DATA_BLOCK "Error_Safety"	// DB 410
AUTHOR : Koenig
VERSION : 0.1
  STRUCT
   Error_09 : BOOL ;	//Emergency stop door 9
   Error_10 : BOOL ;	//Emergency stop door 10
   Error_11 : BOOL ;	//Emergency stop door 11
   Error_12 : BOOL ;	//Emergency stop door 12
   Error_13 : BOOL ;	//Emergency stop door 13
   Error_14 : BOOL ;	//Emergency stop door 14
   Error_15 : BOOL ;	//Emergency stop door 15
   Error_16 : BOOL ;	//Emergency stop door 16
   Error_01 : BOOL ;	//Emergency stop door 1
   Error_02 : BOOL ;	//Emergency stop door 2
   Error_03 : BOOL ;	//Emergency stop door 3
   Error_04 : BOOL ;	//Emergency stop door 4
   Error_05 : BOOL ;	//Emergency stop door 5
   Error_06 : BOOL ;	//Emergency stop door 6
   Error_07 : BOOL ;	//Emergency stop door 7
   Error_08 : BOOL ;	//Emergency stop door 8
   Error_25 : BOOL ;	//Door 9 is unlocked
   Error_26 : BOOL ;	//Door 10 is unlocked
   Error_27 : BOOL ;	//Door 11 is unlocked
   Error_28 : BOOL ;	//Door 12 is unlocked
   Error_29 : BOOL ;	//Door 13 is unlocked
   Error_30 : BOOL ;	//Door 14 is unlocked
   Error_31 : BOOL ;	//Door 15 is unlocked
   Error_32 : BOOL ;	//Door 16 is unlocked
   Error_17 : BOOL ;	//Door 1 is unlocked
   Error_18 : BOOL ;	//Door 2 is unlocked
   Error_19 : BOOL ;	//Door 3 is unlocked
   Error_20 : BOOL ;	//Door 4 is unlocked
   Error_21 : BOOL ;	//Door 5 is unlocked
   Error_22 : BOOL ;	//Door 6 is unlocked
   Error_23 : BOOL ;	//Door 7 is unlocked
   Error_24 : BOOL ;	//Door 8 is unlocked
   Error_41 : BOOL ;
   Error_42 : BOOL ;
   Error_43 : BOOL ;
   Error_44 : BOOL ;
   Error_45 : BOOL ;
   Error_46 : BOOL ;
   Error_47 : BOOL ;
   Error_48 : BOOL ;
   Error_33 : BOOL ;	//Safety light beam 1 tripped
   Error_34 : BOOL ;	//Safety light beam 2 tripped
   Error_35 : BOOL ;	//Safety light beam 3 tripped
   Error_36 : BOOL ;	//Safety light beam 4 tripped
   Error_37 : BOOL ;	//Safety light beam 5 tripped
   Error_38 : BOOL ;	//Safety light beam 6 tripped
   Error_39 : BOOL ;	//Safety light beam 7 tripped
   Error_40 : BOOL ;	//Safety light beam 8 tripped
   Error_57 : BOOL ;
   Error_58 : BOOL ;
   Error_59 : BOOL ;
   Error_60 : BOOL ;
   Error_61 : BOOL ;
   Error_62 : BOOL ;
   Error_63 : BOOL ;
   Error_64 : BOOL ;
   Error_49 : BOOL ;
   Error_50 : BOOL ;	//Emergency stop master
   Error_51 : BOOL ;	//Emergency stop view station #1
   Error_52 : BOOL ;	//Emergency stop view station #2
   Error_53 : BOOL ;	//Emergency stop view station #3
   Error_54 : BOOL ;	//Emergency stop remote crane 1
   Error_55 : BOOL ;	//Emergency stop remote crane 2
   Error_56 : BOOL ;	//Emergency stop main cabinet
   Error_73 : BOOL ;	//CN2 : Relais error emergency mode
   Error_74 : BOOL ;	//CN2 : Relais error bypass remote
   Error_75 : BOOL ;	//CN2 : Relais error fast stop regulator bridge
   Error_76 : BOOL ;	//CN2 : Relais error fast stop regulator trolley
   Error_77 : BOOL ;	//CN2 : Relais error fast stop regulator lift
   Error_78 : BOOL ;	//CN2 : Relais error fast stop regulator width 1
   Error_79 : BOOL ;	//CN2 : Relais error fast stop regulator width 2
   Error_80 : BOOL ;
   Error_65 : BOOL ;	//CN1 : Relais error emergency mode
   Error_66 : BOOL ;	//CN1 : Relais error bypass remote
   Error_67 : BOOL ;	//CN1 : Relais error fast stop regulator bridge
   Error_68 : BOOL ;	//CN1 : Relais error fast stop regulator trolley
   Error_69 : BOOL ;	//CN1 : Relais error fast stop regulator lift
   Error_70 : BOOL ;	//CN1 : Relais error fast stop regulator width 1
   Error_71 : BOOL ;	//CN1 : Relais error fast stop regulator width 2
   Error_72 : BOOL ;
   Error_89 : BOOL ;	//CN2 : no release fast speed bridge
   Error_90 : BOOL ;	//CN2 : no release bridge
   Error_91 : BOOL ;	//CN2 : no release trolley
   Error_92 : BOOL ;	//CN2 : no release lift
   Error_93 : BOOL ;	//CN2 : no release width 1
   Error_94 : BOOL ;	//CN2 : no release width 2
   Error_95 : BOOL ;	//CN2 : no release safety bar
   Error_96 : BOOL ;
   Error_81 : BOOL ;	//CN1 : no release fast speed bridge
   Error_82 : BOOL ;	//CN1 : no release bridge
   Error_83 : BOOL ;	//CN1 : no release trolley
   Error_84 : BOOL ;	//CN1 : no release lift
   Error_85 : BOOL ;	//CN1 : no release width 1
   Error_86 : BOOL ;	//CN1 : no release width 2
   Error_87 : BOOL ;	//CN1 : no release safety bar
   Error_88 : BOOL ;
   Error_105 : BOOL ;	//CN2 : Invalid safety position
   Error_106 : BOOL ;	//CN2 : Invalid safe speed
   Error_107 : BOOL ;	//CN2 : Invalid max speed
   Error_108 : BOOL ;	//CN2 : Safety position difference
   Error_109 : BOOL ;	//CN2 : Signal fault safety closed
   Error_110 : BOOL ;	//CN2 : Invalid operation mode
   Error_111 : BOOL ;	//CN2 : Emergency mode
   Error_112 : BOOL ;	//CN2 : Brake resistors are not OK
   Error_97 : BOOL ;	//CN1 : Invalid safety position
   Error_98 : BOOL ;	//CN1 : Invalid safe speed
   Error_99 : BOOL ;	//CN1 : Invalid max speed
   Error_100 : BOOL ;	//CN1 : Safety position difference
   Error_101 : BOOL ;	//CN1 : Signal fault safety closed
   Error_102 : BOOL ;	//CN1 : Invalid operation mode
   Error_103 : BOOL ;	//CN1 : Emergency mode
   Error_104 : BOOL ;	//CN1 : Brake resistors are not OK
   Error_121 : BOOL ;	//CN2 : Automatic Mode
   Error_122 : BOOL ;	//CN2 : Bypass active
   Error_123 : BOOL ;	//CN2 : Emergency Mode
   Error_124 : BOOL ;	//CN2 : Maintenance
   Error_125 : BOOL ;	//CN2 : crane not on maintenance position
   Error_126 : BOOL ;
   Error_127 : BOOL ;
   Error_128 : BOOL ;
   Error_113 : BOOL ;	//CN1 : Automatic Mode
   Error_114 : BOOL ;	//CN1 : Bypass active
   Error_115 : BOOL ;	//CN1 : Emergency Mode
   Error_116 : BOOL ;	//CN1 : Maintenance
   Error_117 : BOOL ;	//CN1 : crane not on maintenance position
   Error_118 : BOOL ;
   Error_119 : BOOL ;
   Error_120 : BOOL ;
   Error_137 : BOOL ;	//CN2 : Wago unit #1 disturbed
   Error_138 : BOOL ;	//CN2 : Wago unit #2 disturbed
   Error_139 : BOOL ;	//CN2 : Wago unit #3 disturbed
   Error_140 : BOOL ;	//CN2 : Wago unit #4 disturbed
   Error_141 : BOOL ;	//CN2 : Wago unit #5 disturbed
   Error_142 : BOOL ;
   Error_143 : BOOL ;
   Error_144 : BOOL ;
   Error_129 : BOOL ;	//CN1 : Wago unit #1 disturbed
   Error_130 : BOOL ;	//CN1 : Wago unit #2 disturbed
   Error_131 : BOOL ;	//CN1 : Wago unit #3 disturbed
   Error_132 : BOOL ;	//CN1 : Wago unit #4 disturbed
   Error_133 : BOOL ;	//CN1 : Wago unit #5 disturbed
   Error_134 : BOOL ;
   Error_135 : BOOL ;
   Error_136 : BOOL ;
   Error_153 : BOOL ;	//CB : Wago unit #9 disturbed
   Error_154 : BOOL ;	//CB : Wago unit #10 disturbed
   Error_155 : BOOL ;	//CB : Wago unit #11 disturbed
   Error_156 : BOOL ;	//CB : Wago unit #12 disturbed
   Error_157 : BOOL ;	//CB : Wago unit #13 disturbed
   Error_158 : BOOL ;	//CB : Wago unit #14 disturbed
   Error_159 : BOOL ;	//CB : Wago unit #15 disturbed
   Error_160 : BOOL ;	//CB : Wago unit #16 disturbed
   Error_145 : BOOL ;	//CB : Wago unit #1 disturbed
   Error_146 : BOOL ;	//CB : Wago unit #2 disturbed
   Error_147 : BOOL ;	//CB : Wago unit #3 disturbed
   Error_148 : BOOL ;	//CB : Wago unit #4 disturbed
   Error_149 : BOOL ;	//CB : Wago unit #5 disturbed
   Error_150 : BOOL ;	//CB : Wago unit #6 disturbed
   Error_151 : BOOL ;	//CB : Wago unit #7 disturbed
   Error_152 : BOOL ;	//CB : Wago unit #8 disturbed
   Error_169 : BOOL ;	//CR2 : Wago unit #1 disturbed
   Error_170 : BOOL ;	//CR2 : Wago unit #2 disturbed
   Error_171 : BOOL ;	//CR2 : Wago unit #3 disturbed
   Error_172 : BOOL ;	//CR2 : Wago unit #4 disturbed
   Error_173 : BOOL ;
   Error_174 : BOOL ;
   Error_175 : BOOL ;
   Error_176 : BOOL ;
   Error_161 : BOOL ;	//CR1 : Wago unit #1 disturbed
   Error_162 : BOOL ;	//CR1 : Wago unit #2 disturbed
   Error_163 : BOOL ;	//CR1 : Wago unit #3 disturbed
   Error_164 : BOOL ;	//CR1 : Wago unit #4 disturbed
   Error_165 : BOOL ;
   Error_166 : BOOL ;
   Error_167 : BOOL ;
   Error_168 : BOOL ;
   Error_185 : BOOL ;	//MB1 : Wago unit #1 disturbed
   Error_186 : BOOL ;	//MB1 : Wago unit #2 disturbed
   Error_187 : BOOL ;	//MB1 : Wago unit #3 disturbed
   Error_188 : BOOL ;	//MB1 : Wago unit #4 disturbed
   Error_189 : BOOL ;	//SU1 : Wago unit #1 disturbed
   Error_190 : BOOL ;	//SU1 : Wago unit #2 disturbed
   Error_191 : BOOL ;	//SU2 : Wago unit #1 disturbed
   Error_192 : BOOL ;	//SU2 : Wago unit #2 disturbed
   Error_177 : BOOL ;	//CS1 : Wago unit #1 disturbed
   Error_178 : BOOL ;	//CS1 : Wago unit #2 disturbed
   Error_179 : BOOL ;	//CS1 : Wago unit #3 disturbed
   Error_180 : BOOL ;	//CS1 : Wago unit #4 disturbed
   Error_181 : BOOL ;	//CS1 : Wago unit #5 disturbed
   Error_182 : BOOL ;	//CS1 : Wago unit #6 disturbed
   Error_183 : BOOL ;
   Error_184 : BOOL ;
  END_STRUCT ;	
BEGIN
   Error_07 := TRUE;
   Error_137 := TRUE;
   Error_138 := TRUE;
   Error_139 := TRUE;
   Error_140 := TRUE;
   Error_153 := TRUE;
   Error_161 := TRUE;
   Error_185 := TRUE;
   Error_177 := TRUE;
   Error_178 := TRUE;
   Error_179 := TRUE;
   Error_180 := TRUE;
   Error_181 := TRUE;
END_DATA_BLOCK

// DB 450: know-how protected block, not included

// DB 451: know-how protected block, not included

// DB 545: know-how protected block, not included

// DB 546: know-how protected block, not included

// DB 547: know-how protected block, not included

// DB 548: know-how protected block, not included

// DB 549: know-how protected block, not included

// DB 550: know-how protected block, not included

// DB 551: know-how protected block, not included

// DB 552: know-how protected block, not included

// DB 553: know-how protected block, not included

// DB 554: know-how protected block, not included

// DB 555: know-how protected block, not included

// DB 556: know-how protected block, not included

// DB 557: know-how protected block, not included

// DB 558: know-how protected block, not included

// DB 559: know-how protected block, not included

// DB 560: know-how protected block, not included

// DB 561: know-how protected block, not included

// DB 562: know-how protected block, not included

DATA_BLOCK "F_IO"	// DB 690
AUTHOR : Koenig
VERSION : 0.1
  STRUCT
   BRI_EStop : BOOL ;
   BRI_FB_FastStop : BOOL ;
   BRI_FB_EStop_CH1 : BOOL ;
   BRI_FB_EStop_CH2 : BOOL ;
   BRI_Input_04 : BOOL ;
   BRI_Input_05 : BOOL ;
   BRI_Input_06 : BOOL ;
   BRI_Input_07 : BOOL ;
   BRI_TRO_inParkPos_CH1 : BOOL ;
   BRI_TRO_inParkPos_CH2 : BOOL ;
   BRI_Brake_OK : BOOL ;
   BRI_Input_11 : BOOL ;
   BRI_Input_12 : BOOL ;
   BRI_Input_13 : BOOL ;
   BRI_Input_14 : BOOL ;
   BRI_HardwareOK : BOOL ;
   TRO_Spare_DI_35_0 : BOOL ;
   TRO_Spare_DI_35_1 : BOOL ;
   TRO_FB_FastStop_LIF : BOOL ;
   TRO_FB_FastStop_TRO : BOOL ;
   TRO_FB_TastStop_TEL : BOOL ;
   TRO_Spare_DI_40_1 : BOOL ;
   TRO_FB_Estop_CH1 : BOOL ;
   TRO_FB_Estop_CH2 : BOOL ;
   TRO_EStop : BOOL ;
   TRO_Brakes_OK : BOOL ;
   TRO_Spare_DI_45_2 : BOOL ;
   TRO_Spare_DI_45_3 : BOOL ;
   TRO_Input_12 : BOOL ;
   TRO_Input_13 : BOOL ;
   TRO_Input_14 : BOOL ;
   TRO_HardwareOK : BOOL ;
   LIF_Overl_L_NC : BOOL ;
   LIF_Overl_R_NC : BOOL ;
   LIF_Slap_L_NC : BOOL ;
   LIF_Slap_R_NC : BOOL ;
   LIF_Input_04 : BOOL ;
   LIF_Input_05 : BOOL ;
   LIF_Input_06 : BOOL ;
   LIF_Input_07 : BOOL ;
   LIF_Input_08 : BOOL ;
   LIF_Input_09 : BOOL ;
   LIF_Input_10 : BOOL ;
   LIF_Input_11 : BOOL ;
   LIF_Input_12 : BOOL ;
   LIF_Input_13 : BOOL ;
   LIF_Input_14 : BOOL ;
   LIF_HardwareOK : BOOL ;
   CB1_FastStop_Gate_CH1 : BOOL ;
   CB1_FastStop_Gate_CH2 : BOOL ;
   CB1_SPARE_DI220_2 : BOOL ;
   CB1_SPARE_DI220_3 : BOOL ;
   CB1_SPARE_DI225_0 : BOOL ;
   CB1_FastStop : BOOL ;
   CB1_Mode_Auto : BOOL ;
   CB1_Mode_Service : BOOL ;
   CB1_LS1_Door_CH1 : BOOL ;
   CB1_LS1_Door_CH2 : BOOL ;
   CB1_LS2_Door_CH1 : BOOL ;
   CB1_LS2_Door_CH2 : BOOL ;
   CB1_LS3_Door_CH1 : BOOL ;
   CB1_LS3_Door_CH2 : BOOL ;
   CB1_ServiceDoor1_CH1 : BOOL ;
   CB1_ServiceDoor1_CH2 : BOOL ;
   CB1_ServiceDoor2_CH1 : BOOL ;
   CB1_ServiceDoor2_CH2 : BOOL ;
   CB1_ServiceDoor3_CH1 : BOOL ;
   CB1_ServiceDoor3_CH2 : BOOL ;
   CB1_ServiceDoor4_CH1 : BOOL ;
   CB1_ServiceDoor4_CH2 : BOOL ;
   CB1_EStop_Buttons_CH1 : BOOL ;
   CB1_EStop_Buttons_CH2 : BOOL ;
   CB1_EStop_Doors_CH1 : BOOL ;
   CB1_EStop_Doors_CH2 : BOOL ;
   CB1_Service_CH1 : BOOL ;
   CB1_Service_CH2 : BOOL ;
   CB1_Bypass_CH1 : BOOL ;
   CB1_Bypass_CH2 : BOOL ;
   CB1_Auto_ON : BOOL ;
   CB1_SPARE_DI240_7 : BOOL ;
   CB1_PowerON_1 : BOOL ;
   CB1_PowerON_2 : BOOL ;
   CB1_SPARE_DO220_2 : BOOL ;
   CB1_SPARE_DO220_3 : BOOL ;
   CB1_SPARE_DO225_0 : BOOL ;
   CB1_SPARE_DO225_1 : BOOL ;
   CB1_SPARE_DO225_2 : BOOL ;
   CB1_SPARE_DO225_3 : BOOL ;
   MB1_Power_ON_1 : BOOL ;
   MB1_Power_ON_2 : BOOL ;
   MB1_ESTOP_1 : BOOL ;
   MB1_ESTOP_2 : BOOL ;
   MB1_HardwareOK : BOOL ;
   MB1_FB_Power_ON : BOOL ;
   MB1_INPUT_07 : BOOL ;
   MB1_INPUT_08 : BOOL ;
   SU1_HardwareOK : BOOL ;
   SU1_Scanner_Plus_OK : BOOL ;
   SU1_Scanner_Minus_OK : BOOL ;
   SU1_ReglerPowerON : BOOL ;
   SU1_INPUT_05 : BOOL ;
   SU1_INPUT_06 : BOOL ;
   SU1_INPUT_07 : BOOL ;
   SU1_INPUT_08 : BOOL ;
   SU2_HardwareOK : BOOL ;
   SU2_Scanner_Plus_OK : BOOL ;
   SU2_Scanner_Minus_OK : BOOL ;
   SU2_ReglerPowerON : BOOL ;
   SU2_INPUT_05 : BOOL ;
   SU2_INPUT_06 : BOOL ;
   SU2_INPUT_07 : BOOL ;
   SU2_INPUT_08 : BOOL ;
  END_STRUCT ;	
BEGIN
   BRI_EStop := TRUE;
   BRI_FB_EStop_CH2 := TRUE;
   BRI_Input_04 := TRUE;
   TRO_Brakes_OK := TRUE;
   LIF_Overl_L_NC := TRUE;
   LIF_Overl_R_NC := TRUE;
   LIF_Slap_L_NC := TRUE;
   LIF_Slap_R_NC := TRUE;
   CB1_Mode_Auto := TRUE;
   CB1_EStop_Buttons_CH2 := TRUE;
   CB1_EStop_Doors_CH1 := TRUE;
   CB1_EStop_Doors_CH2 := TRUE;
   CB1_Service_CH1 := TRUE;
   CB1_Service_CH2 := TRUE;
   CB1_Auto_ON := TRUE;
   CB1_SPARE_DI240_7 := TRUE;
   CB1_PowerON_1 := TRUE;
   CB1_PowerON_2 := TRUE;
   CB1_SPARE_DO220_2 := TRUE;
   CB1_SPARE_DO220_3 := TRUE;
   CB1_SPARE_DO225_0 := TRUE;
   CB1_SPARE_DO225_1 := TRUE;
   CB1_SPARE_DO225_2 := TRUE;
   CB1_SPARE_DO225_3 := TRUE;
   MB1_FB_Power_ON := TRUE;
END_DATA_BLOCK

DATA_BLOCK "F_Position"	// DB 695
VERSION : 0.1
  STRUCT
   TR_POS_CM : INT ;
   CAR1_ActualPos : INT ;
   CAR2_ActualPos : INT ;
   TR_POS_CM_REL : INT ;
   Spare02 : INT ;
   BR_Area : INT ;
   TR_Area : INT ;
   Spare03 : INT ;
   Spare04 : INT ;
   Spare05 : INT ;
   BR01_TR0209_Start : INT ;	//2000 - 5000
   BR01_TR0209_Stop : INT ;
   BR02_TR0209_Start : INT ;	//5000 - 8000
   BR02_TR0209_Stop : INT ;
   BR03_TR0209_Start : INT ;	//8000 - 11000
   BR03_TR0209_Stop : INT ;
   BR04_TR0209_Start : INT ;	//11000 - 14000
   BR04_TR0209_Stop : INT ;
   BR05_TR0209_Start : INT ;	//14000 - 17000
   BR05_TR0209_Stop : INT ;
   BR06_TR0209_Start : INT ;	//17000 - 20000
   BR06_TR0209_Stop : INT ;
   BR07_TR0209_Start : INT ;	//20000 - 23000
   BR07_TR0209_Stop : INT ;
   BR08_TR0209_Start : INT ;	//23000 - 26000
   BR08_TR0209_Stop : INT ;
   BR09_TR0209_Start : INT ;	//26000 - 29000
   BR09_TR0209_Stop : INT ;
   BR10_TR0209_Start : INT ;	//29000 - 32000
   BR10_TR0209_Stop : INT ;
   BR11_TR0209_Start : INT ;	//38000 - 39000
   BR11_TR0209_Stop : INT ;
   BR01_TR11_Start : INT ;	//33000 - 34000
   BR01_TR11_Stop : INT ;
   BR02_TR11_Start : INT ;	//34000 - 35000
   BR02_TR11_Stop : INT ;
   BR03_TR11_Start : INT ;	//35000 - 36000
   BR03_TR11_Stop : INT ;
   BR04_TR11_Start : INT ;	//36000 - 37000
   BR04_TR11_Stop : INT ;
   BR05_TR11_Start : INT ;	//37000 - 38000
   BR05_TR11_Stop : INT ;
   BR06_TR11_Start : INT ;	//xxx
   BR06_TR11_Stop : INT ;
   BR07_TR11_Start : INT ;	//xxx
   BR07_TR11_Stop : INT ;
   BR08_TR11_Start : INT ;	//xxx
   BR08_TR11_Stop : INT ;
   BR09_TR11_Start : INT ;	//xxx
   BR09_TR11_Stop : INT ;
   BR10_TR11_Start : INT ;	//xxx
   BR10_TR11_Stop : INT ;
   CAR01_TR01_Start : INT ;	//0 - 1000
   CAR01_TR01_Stop : INT ;
   CAR02_TR10_Start : INT ;	//32000 - 33000
   CAR02_TR10_Stop : INT ;
  END_STRUCT ;	
BEGIN
   TR_POS_CM := 16021;
   TR_POS_CM_REL := 2401;
   BR_Area := 5;
   TR_Area := 8;
   BR01_TR0209_Start := 1800;
   BR01_TR0209_Stop := 4500;
   BR02_TR0209_Start := 4800;
   BR02_TR0209_Stop := 7500;
   BR03_TR0209_Start := 7800;
   BR03_TR0209_Stop := 10500;
   BR04_TR0209_Start := 10800;
   BR04_TR0209_Stop := 13500;
   BR05_TR0209_Start := 13800;
   BR05_TR0209_Stop := 16500;
   BR06_TR0209_Start := 16800;
   BR06_TR0209_Stop := 19500;
   BR07_TR0209_Start := 19800;
   BR07_TR0209_Stop := 22500;
   BR08_TR0209_Start := 22800;
   BR08_TR0209_Stop := 25500;
   BR09_TR0209_Start := 25800;
   BR09_TR0209_Stop := 28500;
   BR10_TR0209_Start := 28800;
   BR10_TR0209_Stop := 31500;
   CAR01_TR01_Stop := 1000;
   CAR02_TR10_Start := 31900;
   CAR02_TR10_Stop := 32380;
END_DATA_BLOCK

DATA_BLOCK "F_GBL_RECV"	// DB 750
AUTHOR : Koenig
FAMILY : COM_DBS7
VERSION : 0.1
  STRUCT
   Signal01 : BOOL ;	//Automatic mode
   Signal02 : BOOL ;	//Bypass
   Signal03 : BOOL ;	//Reset
   Signal04 : BOOL ;	//NO E-Stop
   Signal05 : BOOL ;	//Start Automatic
   Signal06 : BOOL ;	//Release drive
   Signal07 : BOOL ;	//Release drive fast
   Signal08 : BOOL ;	//Service mode
   Signal09 : BOOL ;
   Signal10 : BOOL ;	//Safety area rack OK
   Signal11 : BOOL ;
   Signal12 : BOOL ;
   Signal13 : BOOL ;
   Signal14 : BOOL ;
   Signal15 : BOOL ;
   Signal16 : BOOL ;
   Signal17 : BOOL ;
   Signal18 : BOOL ;
   Signal19 : BOOL ;
   Signal20 : BOOL ;
   Signal21 : BOOL ;
   Signal22 : BOOL ;
   Signal23 : BOOL ;
   Signal24 : BOOL ;
   Signal25 : BOOL ;
   Signal26 : BOOL ;
   Signal27 : BOOL ;
   Signal28 : BOOL ;
   Signal29 : BOOL ;
   Signal30 : BOOL ;
   Signal31 : BOOL ;
   Signal32 : BOOL ;
   Value01 : INT ;	//Position carrier 1
   Value02 : INT ;	//Position carrier 2
   Value03 : INT ;
   Value04 : INT ;
  END_STRUCT ;	
BEGIN
   Signal01 := TRUE;
   Signal04 := TRUE;
   Signal06 := TRUE;
   Signal07 := TRUE;
   Signal10 := TRUE;
   Value01 := 5;
   Value02 := 3;
END_DATA_BLOCK

// DB 751: know-how protected block, not included

DATA_BLOCK "F_GBL_SEND"	// DB 752
AUTHOR : Koenig
FAMILY : COM_DBS7
VERSION : 0.1
  STRUCT
   Signal01 : BOOL ;	//Trolley is in position (unsafe)
   Signal02 : BOOL ;	//Teleskope is in center (unsafe)
   Signal03 : BOOL ;	//Teleskope is in rear (unsafe)
   Signal04 : BOOL ;	//Teleskope is in front (unsafe)
   Signal05 : BOOL ;	//Lift in top position (unsafe)
   Signal06 : BOOL ;	//Lift in over position (unsafe)
   Signal07 : BOOL ;	//Lift in under position (unsafe)
   Signal08 : BOOL ;	//Lift in top position (unsafe, sensor)
   Signal09 : BOOL ;
   Signal10 : BOOL ;
   Signal11 : BOOL ;
   Signal12 : BOOL ;
   Signal13 : BOOL ;
   Signal14 : BOOL ;
   Signal15 : BOOL ;
   Signal16 : BOOL ;
   Value01 : INT ;	//Area Trolley (no.)
   Value02 : INT ;	//Area Lift (no.)
   Value03 : INT ;	//Area Bridge (no.)
   Value04 : INT ;	//Trolley Axis value
   Value05 : INT ;	//Trolley Axis releative 2-9 / 11
  END_STRUCT ;	
BEGIN
   Signal01 := TRUE;
   Signal02 := TRUE;
   Value01 := 8;
   Value02 := 6;
   Value03 := 5;
   Value04 := 16021;
   Value05 := 2401;
END_DATA_BLOCK

// DB 753: know-how protected block, not included

DATA_BLOCK "IDB_Axis_Position"	// DB 800
AUTHOR : BRO
VERSION : 0.1
"Axis_Position"
BEGIN
END_DATA_BLOCK

DATA_BLOCK "IDB_WagoiPar_Rack"	// DB 901
AUTHOR : JPR
FAMILY : WAGOiPar
VERSION : 0.0
"WAGO_iPar_UDL_4_Mod"
BEGIN
END_DATA_BLOCK

DATA_BLOCK "IDB_WagoiPar_BRI"	// DB 920
AUTHOR : JPR
FAMILY : WAGOiPar
VERSION : 0.0
"WAGO_iPar_UDL_4_Mod"
BEGIN
END_DATA_BLOCK

DATA_BLOCK "IDB_WagoiPar_TRO"	// DB 921
AUTHOR : JPR
FAMILY : WAGOiPar
VERSION : 0.0
"WAGO_iPar_UDL_4_Mod"
BEGIN
END_DATA_BLOCK

DATA_BLOCK "IDB_WagoiPar_LIF"	// DB 922
AUTHOR : JPR
FAMILY : WAGOiPar
VERSION : 0.0
"WAGO_iPar_UDL_4_Mod"
BEGIN
END_DATA_BLOCK

DATA_BLOCK "DB_iPar_Diag"	// DB 930
AUTHOR : JPR
FAMILY : WAGOiPar
VERSION : 0.0
"DiagPROFIsafe_V2_iPar"
BEGIN
END_DATA_BLOCK

DATA_BLOCK "DIAG_PROFI_V2_iPar"	// DB 931
TITLE = Vorlage Datenbaustein zur Ablage der Diagnosedaten FB101
//Template data block used in combination with FB101
//
AUTHOR : JPR
FAMILY : WAGOiPar
NAME : iParInfD
VERSION : 1.0
  STRUCT
   versionInfo_1 : INT  := 101;	//version info main
   versionInfo_2 : WORD  := W#16#100;	//version info release
   spare_4 : WORD ;
   fctReqTimeout : INT  := 6000;	//function request timeout (default 6000; av.cycle plc 5 ms - timeout 30 s)
   dsvLength : INT  := 20;	//lenght of storage data
   maxModules : INT  := 1;	//amount PROFIsafe modules FB101
   adr_module_1 : INT ;	//I/O address module 1
   adr_module_2 : INT ;	//I/O address module 2
   adr_module_3 : INT ;	//I/O address module 3
   adr_module_4 : INT ;	//I/O address module 4
   adr_module_5 : INT ;	//I/O address module 5
   adr_module_6 : INT ;	//I/O address module 6
   adr_module_7 : INT ;	//I/O address module 7
   adr_module_8 : INT ;	//I/O address module 8
   adr_module_9 : INT ;	//I/O address module 9
   adr_module_10 : INT ;	//I/O address module 10
   adr_module_11 : INT ;	//I/O address module 11
   adr_module_12 : INT ;	//I/O address module 12
   spare_34 : WORD ;
   spare_36 : WORD ;
   Init_Date : DATE ;	//startup date application slave
   InitTime : TIME_OF_DAY ;	//startup time application slave
   spare_46 : WORD ;
   spare_48 : WORD ;
   actDateCyle1 : DATE ;	//actual system date of cycle
   actTimeCyle1 : TIME_OF_DAY ;	//actual system time of cycle
   spare_56 : WORD ;
   spare_58 : WORD ;
   QBAD_moduleActive : DWORD ;	//info QBAD at PROFIsafe module active
   ACK_REQ_moduleActive : DWORD ;	//info ACK_REQ at PROFIsafe module active
   READ_DIAG_REQ_module : DWORD ;	//info READ_DIAG_REQ at PROFIsafe module active
   spare_72 : WORD ;
   spare_74 : WORD ;
   check_cfg_done : DWORD ;	//info check cfg done
   read_diag_done : DWORD ;	//info read diag done
   spare_84 : WORD ;
   spare_86 : WORD ;
   resFctReq_ok : DWORD ;	//response function request ok - "bit per module"
   resFctReq_error : DWORD ;	//response function request error - "bit per module"
   spare_96 : WORD ;
   spare_98 : WORD ;
   cmdCtrl_FB101_1 : WORD ;	//cmd / ctrl information FB101
   comCountStart_1 : WORD ;	//comCountStart indication 1
   mod_type_1 : WORD ;	//module type 1
   mod_version_1 : WORD ;	//module version 1
   spare_108 : WORD ;
   state_SFB52_1 : DWORD ;	//state SFB52 module 1
   spare_114 : WORD ;
   spare_116 : WORD ;
   error_date_mod_1 : DATE ;	//error date module 1
   error_time_mod_1 : TIME_OF_DAY ;	//error time module 1
   error_info_mod_1 : WORD ;	//error info read values module 1
   error_F_Module_mod_1 : WORD ;	//error safety module module 1
   error_F_DI_1_mod_1 : WORD ;	//error safety input 1 module 1
   error_F_DI_2_mod_1 : WORD ;	//error safety input 2 module 1
   error_F_DI_3_mod_1 : WORD ;	//error safety input 3 module 1
   error_F_DI_4_mod_1 : WORD ;	//error safety input 4 module 1
   error_F_DI_5_mod_1 : WORD ;	//error safety input 5 module 1
   error_F_DI_6_mod_1 : WORD ;	//error safety input 6 module 1
   error_F_DI_7_mod_1 : WORD ;	//error safety input 7 module 1
   error_F_DI_8_mod_1 : WORD ;	//error safety input 8 module 1
   error_F_DO_1_mod_1 : WORD ;	//error safety output 1 module 1
   error_F_DO_2_mod_1 : WORD ;	//error safety output 2 module 1
   error_F_DO_3_mod_1 : WORD ;	//error safety output 3 module 1
   error_F_DO_4_mod_1 : WORD ;	//error safety output 4 module 1
   error_F_Mod_R48_mod_1 : WORD ;	//error safety R48 module 1
   error_F_Mod_R49_mod_1 : WORD ;	//error safety R49 module 1
   error_F_Mod_R50_mod_1 : WORD ;	//error safety R50 module 1
   error_F_Mod_R51_mod_1 : WORD ;	//error safety R51 module 1
   error_F_Mod_R52_mod_1 : WORD ;	//error safety R52 module 1
   error_F_Mod_R53_mod_1 : WORD ;	//error safety R53 module 1
   error_F_Mod_R54_mod_1 : WORD ;	//error safety R54 module 1
   error_F_Mod_R55_mod_1 : WORD ;	//error safety R55 module 1
   F_Per_DB_B3_mod_1 : WORD ;	//state F-Periphery DB module 1
   spare_170 : WORD ;
   spare_172 : WORD ;
   spare_174 : WORD ;
   spare_176 : WORD ;
   spare_178 : WORD ;
   cmdCtrl_FB101_2 : WORD ;	//cmd / ctrl information FB101
   comCountStart_2 : WORD ;	//comCountStart indication
   mod_type_2 : WORD ;	//module type
   mod_version_2 : WORD ;	//module version
   spare_188 : WORD ;
   state_SFB52_2 : DWORD ;	//state SFB52 module
   spare_194 : WORD ;
   spare_196 : WORD ;
   error_date_mod_2 : DATE ;	//error date module 2
   error_time_mod_2 : TIME_OF_DAY ;	//error time module 2
   error_info_mod_2 : WORD ;	//error info read values module 2
   error_F_Module_mod_2 : WORD ;	//error safety module module 2
   error_F_DI_1_mod_2 : WORD ;	//error safety input 1 module 2
   error_F_DI_2_mod_2 : WORD ;	//error safety input 2 module 2
   error_F_DI_3_mod_2 : WORD ;	//error safety input 3 module 2
   error_F_DI_4_mod_2 : WORD ;	//error safety input 4 module 2
   error_F_DI_5_mod_2 : WORD ;	//error safety input 5 module 2
   error_F_DI_6_mod_2 : WORD ;	//error safety input 6 module 2
   error_F_DI_7_mod_2 : WORD ;	//error safety input 7 module 2
   error_F_DI_8_mod_2 : WORD ;	//error safety input 8 module 2
   error_F_DO_1_mod_2 : WORD ;	//error safety output 1 module 2
   error_F_DO_2_mod_2 : WORD ;	//error safety output 2 module 2
   error_F_DO_3_mod_2 : WORD ;	//error safety output 3 module 2
   error_F_DO_4_mod_2 : WORD ;	//error safety output 4 module 2
   error_F_Mod_R48_mod_2 : WORD ;	//error safety R48 module 2
   error_F_Mod_R49_mod_2 : WORD ;	//error safety R49 module 2
   error_F_Mod_R50_mod_2 : WORD ;	//error safety R50 module 2
   error_F_Mod_R51_mod_2 : WORD ;	//error safety R51 module 2
   error_F_Mod_R52_mod_2 : WORD ;	//error safety R52 module 2
   error_F_Mod_R53_mod_2 : WORD ;	//error safety R53 module 2
   error_F_Mod_R54_mod_2 : WORD ;	//error safety R54 module 2
   error_F_Mod_R55_mod_2 : WORD ;	//error safety R55 module 2
   F_Per_DB_B3_mod_2 : WORD ;	//state F-Periphery DB module 2
   spare_250 : WORD ;
   spare_252 : WORD ;
   spare_254 : WORD ;
   spare_256 : WORD ;
   spare_258 : WORD ;
   cmdCtrl_FB101_3 : WORD ;	//cmd / ctrl information FB101
   comCountStart_3 : WORD ;	//comCountStart indication
   mod_type_3 : WORD ;	//module type
   mod_version_3 : WORD ;	//module version
   spare_268 : WORD ;
   state_SFB52_3 : DWORD ;	//state SFB52 module
   spare_274 : WORD ;
   spare_276 : WORD ;
   error_date_mod_3 : DATE ;	//error date module 3
   error_time_mod_3 : TIME_OF_DAY ;	//error time module 3
   error_info_mod_3 : WORD ;	//error info read values module 3
   error_F_Module_mod_3 : WORD ;	//error safety module module 3
   error_F_DI_1_mod_3 : WORD ;	//error safety input 1 module 3
   error_F_DI_2_mod_3 : WORD ;	//error safety input 2 module 3
   error_F_DI_3_mod_3 : WORD ;	//error safety input 3 module 3
   error_F_DI_4_mod_3 : WORD ;	//error safety input 4 module 3
   error_F_DI_5_mod_3 : WORD ;	//error safety input 5 module 3
   error_F_DI_6_mod_3 : WORD ;	//error safety input 6 module 3
   error_F_DI_7_mod_3 : WORD ;	//error safety input 7 module 3
   error_F_DI_8_mod_3 : WORD ;	//error safety input 8 module 3
   error_F_DO_1_mod_3 : WORD ;	//error safety output 1 module 3
   error_F_DO_2_mod_3 : WORD ;	//error safety output 2 module 3
   error_F_DO_3_mod_3 : WORD ;	//error safety output 3 module 3
   error_F_DO_4_mod_3 : WORD ;	//error safety output 4 module 3
   error_F_Mod_R48_mod_3 : WORD ;	//error safety R48 module 3
   error_F_Mod_R49_mod_3 : WORD ;	//error safety R49 module 3
   error_F_Mod_R50_mod_3 : WORD ;	//error safety R50 module 3
   error_F_Mod_R51_mod_3 : WORD ;	//error safety R51 module 3
   error_F_Mod_R52_mod_3 : WORD ;	//error safety R52 module 3
   error_F_Mod_R53_mod_3 : WORD ;	//error safety R53 module 3
   error_F_Mod_R54_mod_3 : WORD ;	//error safety R54 module 3
   error_F_Mod_R55_mod_3 : WORD ;	//error safety R55 module 3
   F_Per_DB_B3_mod_3 : WORD ;	//state F-Periphery DB module 3
   spare_330 : WORD ;
   spare_332 : WORD ;
   spare_334 : WORD ;
   spare_336 : WORD ;
   spare_338 : WORD ;
   cmdCtrl_FB101_4 : WORD ;	//cmd / ctrl information FB101
   comCountStart_4 : WORD ;	//comCountStart indication
   mod_type4 : WORD ;	//module type
   mod_version_4 : WORD ;	//module version
   spare_348 : WORD ;
   state_SFB52_4 : DWORD ;	//state SFB52 module
   spare_354 : WORD ;
   spare_356 : WORD ;
   error_date_mod_4 : DATE ;	//error date module 4
   error_time_mod_4 : TIME_OF_DAY ;	//error time module 4
   error_info_mod_4 : WORD ;	//error info read values module 4
   error_F_Module_mod_4 : WORD ;	//error safety module module 4
   error_F_DI_1_mod_4 : WORD ;	//error safety input 1 module 4
   error_F_DI_2_mod_4 : WORD ;	//error safety input 2 module 4
   error_F_DI_3_mod_4 : WORD ;	//error safety input 3 module 4
   error_F_DI_4_mod_4 : WORD ;	//error safety input 4 module 4
   error_F_DI_5_mod_4 : WORD ;	//error safety input 5 module 4
   error_F_DI_6_mod_4 : WORD ;	//error safety input 6 module 4
   error_F_DI_7_mod_4 : WORD ;	//error safety input 7 module 4
   error_F_DI_8_mod_4 : WORD ;	//error safety input 8 module 4
   error_F_DO_1_mod_4 : WORD ;	//error safety output 1 module 4
   error_F_DO_2_mod_4 : WORD ;	//error safety output 2 module 4
   error_F_DO_3_mod_4 : WORD ;	//error safety output 3 module 4
   error_F_DO_4_mod_4 : WORD ;	//error safety output 4 module 4
   error_F_Mod_R48_mod_4 : WORD ;	//error safety R48 module 4
   error_F_Mod_R49_mod_4 : WORD ;	//error safety R49 module 4
   error_F_Mod_R50_mod_4 : WORD ;	//error safety R50 module 4
   error_F_Mod_R51_mod_4 : WORD ;	//error safety R51 module 4
   error_F_Mod_R52_mod_4 : WORD ;	//error safety R52 module 4
   error_F_Mod_R53_mod_4 : WORD ;	//error safety R53 module 4
   error_F_Mod_R54_mod_4 : WORD ;	//error safety R54 module 4
   error_F_Mod_R55_mod_4 : WORD ;	//error safety R55 module 4
   F_Per_DB_B3_mod_4 : WORD ;	//state F-Periphery DB module 4
   spare_410 : WORD ;
   spare_412 : WORD ;
   spare_414 : WORD ;
   spare_416 : WORD ;
   spare_418 : WORD ;
   cmdCtrl_FB101_5 : WORD ;	//cmd / ctrl information FB101
   comCountStart_5 : WORD ;	//comCountStart indication
   mod_type_5 : WORD ;	//module type
   mod_version_5 : WORD ;	//module version
   spare_428 : WORD ;
   state_SFB52_5 : DWORD ;	//state SFB52 module
   spare_434 : WORD ;
   spare_436 : WORD ;
   error_date_mod_5 : DATE ;	//error date module 5
   error_time_mod_5 : TIME_OF_DAY ;	//error time module 5
   error_info_mod_5 : WORD ;	//error info read values module 5
   error_F_Module_mod_5 : WORD ;	//error safety module module 5
   error_F_DI_1_mod_5 : WORD ;	//error safety input 1 module 5
   error_F_DI_2_mod_5 : WORD ;	//error safety input 2 module 5
   error_F_DI_3_mod_5 : WORD ;	//error safety input 3 module 5
   error_F_DI_4_mod_5 : WORD ;	//error safety input 4 module 5
   error_F_DI_5_mod_5 : WORD ;	//error safety input 5 module 5
   error_F_DI_6_mod_5 : WORD ;	//error safety input 6 module 5
   error_F_DI_7_mod_5 : WORD ;	//error safety input 7 module 5
   error_F_DI_8_mod_5 : WORD ;	//error safety input 8 module 5
   error_F_DO_1_mod_5 : WORD ;	//error safety output 1 module 5
   error_F_DO_2_mod_5 : WORD ;	//error safety output 2 module 5
   error_F_DO_3_mod_5 : WORD ;	//error safety output 3 module 5
   error_F_DO_4_mod_5 : WORD ;	//error safety output 4 module 5
   error_F_Mod_R48_mod_5 : WORD ;	//error safety R48 module 5
   error_F_Mod_R49_mod_5 : WORD ;	//error safety R49 module 5
   error_F_Mod_R50_mod_5 : WORD ;	//error safety R50 module 5
   error_F_Mod_R51_mod_5 : WORD ;	//error safety R51 module 5
   error_F_Mod_R52_mod_5 : WORD ;	//error safety R52 module 5
   error_F_Mod_R53_mod_5 : WORD ;	//error safety R53 module 5
   error_F_Mod_R54_mod_5 : WORD ;	//error safety R54 module 5
   error_F_Mod_R55_mod_5 : WORD ;	//error safety R55 module 5
   F_Per_DB_B3_mod_5 : WORD ;	//state F-Periphery DB module 5
   spare_490 : WORD ;
   spare_492 : WORD ;
   spare_494 : WORD ;
   spare_496 : WORD ;
   spare_498 : WORD ;
   cmdCtrl_FB101_6 : WORD ;	//cmd / ctrl information FB101
   comCountStart_6 : WORD ;	//comCountStart indication
   mod_type_6 : WORD ;	//module type
   mod_version_6 : WORD ;	//module version
   spare_508 : WORD ;
   state_SFB52_6 : DWORD ;	//state SFB52 module
   spare_514 : WORD ;
   spare_516 : WORD ;
   error_date_mod_6 : DATE ;	//error date module 6
   error_time_mod_6 : TIME_OF_DAY ;	//error time module 6
   error_info_mod_6 : WORD ;	//error info read values module 6
   error_F_Module_mod_6 : WORD ;	//error safety module module 6
   error_F_DI_1_mod_6 : WORD ;	//error safety input 1 module 6
   error_F_DI_2_mod_6 : WORD ;	//error safety input 2 module 6
   error_F_DI_3_mod_6 : WORD ;	//error safety input 3 module 6
   error_F_DI_4_mod_6 : WORD ;	//error safety input 4 module 6
   error_F_DI_5_mod_6 : WORD ;	//error safety input 5 module 6
   error_F_DI_6_mod_6 : WORD ;	//error safety input 6 module 6
   error_F_DI_7_mod_6 : WORD ;	//error safety input 7 module 6
   error_F_DI_8_mod_6 : WORD ;	//error safety input 8 module 6
   error_F_DO_1_mod_6 : WORD ;	//error safety output 1 module 6
   error_F_DO_2_mod_6 : WORD ;	//error safety output 2 module 6
   error_F_DO_3_mod_6 : WORD ;	//error safety output 3 module 6
   error_F_DO_4_mod_6 : WORD ;	//error safety output 4 module 6
   error_F_Mod_R48_mod_6 : WORD ;	//error safety R48 module 6
   error_F_Mod_R49_mod_6 : WORD ;	//error safety R49 module 6
   error_F_Mod_R50_mod_6 : WORD ;	//error safety R50 module 6
   error_F_Mod_R51_mod_6 : WORD ;	//error safety R51 module 6
   error_F_Mod_R52_mod_6 : WORD ;	//error safety R52 module 6
   error_F_Mod_R53_mod_6 : WORD ;	//error safety R53 module 6
   error_F_Mod_R54_mod_6 : WORD ;	//error safety R54 module 6
   error_F_Mod_R55_mod_6 : WORD ;	//error safety R55 module 6
   F_Per_DB_B3_mod_6 : WORD ;	//state F-Periphery DB module 6
   spare_570 : WORD ;
   spare_572 : WORD ;
   spare_574 : WORD ;
   spare_576 : WORD ;
   spare_578 : WORD ;
   cmdCtrl_FB101_7 : WORD ;	//cmd / ctrl information FB101
   comCountStart_7 : WORD ;	//comCountStart indication
   mod_type_7 : WORD ;	//module type
   mod_version_7 : WORD ;	//module version
   spare_588 : WORD ;
   state_SFB52_7 : DWORD ;	//state SFB52 module
   spare_594 : WORD ;
   spare_596 : WORD ;
   error_date_mod_7 : DATE ;	//error date module 7
   error_time_mod_7 : TIME_OF_DAY ;	//error time module 7
   error_info_mod_7 : WORD ;	//error info read values module 7
   error_F_Module_mod_7 : WORD ;	//error safety module module 7
   error_F_DI_1_mod_7 : WORD ;	//error safety input 1 module 7
   error_F_DI_2_mod_7 : WORD ;	//error safety input 2 module 7
   error_F_DI_3_mod_7 : WORD ;	//error safety input 3 module 7
   error_F_DI_4_mod_7 : WORD ;	//error safety input 4 module 7
   error_F_DI_5_mod_7 : WORD ;	//error safety input 5 module 7
   error_F_DI_6_mod_7 : WORD ;	//error safety input 6 module 7
   error_F_DI_7_mod_7 : WORD ;	//error safety input 7 module 7
   error_F_DI_8_mod_7 : WORD ;	//error safety input 8 module 7
   error_F_DO_1_mod_7 : WORD ;	//error safety output 1 module 7
   error_F_DO_2_mod_7 : WORD ;	//error safety output 2 module 7
   error_F_DO_3_mod_7 : WORD ;	//error safety output 3 module 7
   error_F_DO_4_mod_7 : WORD ;	//error safety output 4 module 7
   error_F_Mod_R48_mod_7 : WORD ;	//error safety R48 module 7
   error_F_Mod_R49_mod_7 : WORD ;	//error safety R49 module 7
   error_F_Mod_R50_mod_7 : WORD ;	//error safety R50 module 7
   error_F_Mod_R51_mod_7 : WORD ;	//error safety R51 module 7
   error_F_Mod_R52_mod_7 : WORD ;	//error safety R52 module 7
   error_F_Mod_R53_mod_7 : WORD ;	//error safety R53 module 7
   error_F_Mod_R54_mod_7 : WORD ;	//error safety R54 module 7
   error_F_Mod_R55_mod_7 : WORD ;	//error safety R55 module 7
   F_Per_DB_B3_mod_7 : WORD ;	//state F-Periphery DB module 7
   spare_650 : WORD ;
   spare_652 : WORD ;
   spare_654 : WORD ;
   spare_656 : WORD ;
   spare_658 : WORD ;
   cmdCtrl_FB101_8 : WORD ;	//cmd / ctrl information FB101
   comCountStart_8 : WORD ;	//comCountStart indication
   mod_type_8 : WORD ;	//module type
   mod_version_8 : WORD ;	//module version
   spare_668 : WORD ;
   state_SFB52_8 : DWORD ;	//state SFB52 module
   spare_674 : WORD ;
   spare_676 : WORD ;
   error_date_mod_8 : DATE ;	//error date module 8
   error_time_mod_8 : TIME_OF_DAY ;	//error time module 8
   error_info_mod_8 : WORD ;	//error info read values module 8
   error_F_Module_mod_8 : WORD ;	//error safety module module 8
   error_F_DI_1_mod_8 : WORD ;	//error safety input 1 module 8
   error_F_DI_2_mod_8 : WORD ;	//error safety input 2 module 8
   error_F_DI_3_mod_8 : WORD ;	//error safety input 3 module 8
   error_F_DI_4_mod_8 : WORD ;	//error safety input 4 module 8
   error_F_DI_5_mod_8 : WORD ;	//error safety input 5 module 8
   error_F_DI_6_mod_8 : WORD ;	//error safety input 6 module 8
   error_F_DI_7_mod_8 : WORD ;	//error safety input 7 module 8
   error_F_DI_8_mod_8 : WORD ;	//error safety input 8 module 8
   error_F_DO_1_mod_8 : WORD ;	//error safety output 1 module 8
   error_F_DO_2_mod_8 : WORD ;	//error safety output 2 module 8
   error_F_DO_3_mod_8 : WORD ;	//error safety output 3 module 8
   error_F_DO_4_mod_8 : WORD ;	//error safety output 4 module 8
   error_F_Mod_R48_mod_8 : WORD ;	//error safety R48 module 8
   error_F_Mod_R49_mod_8 : WORD ;	//error safety R49 module 8
   error_F_Mod_R50_mod_8 : WORD ;	//error safety R50 module 8
   error_F_Mod_R51_mod_8 : WORD ;	//error safety R51 module 8
   error_F_Mod_R52_mod_8 : WORD ;	//error safety R52 module 8
   error_F_Mod_R53_mod_8 : WORD ;	//error safety R53 module 8
   error_F_Mod_R54_mod_8 : WORD ;	//error safety R54 module 8
   error_F_Mod_R55_mod_8 : WORD ;	//error safety R55 module 8
   F_Per_DB_B3_mod_8 : WORD ;	//state F-Periphery DB module 8
   spare_730 : WORD ;
   spare_732 : WORD ;
   spare_734 : WORD ;
   spare_736 : WORD ;
   spare_738 : WORD ;
   cmdCtrl_FB101_9 : WORD ;	//cmd / ctrl information FB101
   comCountStart_9 : WORD ;	//comCountStart indication
   mod_type_9 : WORD ;	//module type
   mod_version_9 : WORD ;	//module version
   spare_748 : WORD ;
   state_SFB52_9 : DWORD ;	//state SFB52 module
   spare_754 : WORD ;
   spare_756 : WORD ;
   error_date_mod_9 : DATE ;	//error date module 9
   error_time_mod_9 : TIME_OF_DAY ;	//error time module 9
   error_info_mod_9 : WORD ;	//error info read values module 9
   error_F_Module_mod_9 : WORD ;	//error safety module module 9
   error_F_DI_1_mod_9 : WORD ;	//error safety input 1 module 9
   error_F_DI_2_mod_9 : WORD ;	//error safety input 2 module 9
   error_F_DI_3_mod_9 : WORD ;	//error safety input 3 module 9
   error_F_DI_4_mod_9 : WORD ;	//error safety input 4 module 9
   error_F_DI_5_mod_9 : WORD ;	//error safety input 5 module 9
   error_F_DI_6_mod_9 : WORD ;	//error safety input 6 module 9
   error_F_DI_7_mod_9 : WORD ;	//error safety input 7 module 9
   error_F_DI_8_mod_9 : WORD ;	//error safety input 8 module 9
   error_F_DO_1_mod_9 : WORD ;	//error safety output 1 module 9
   error_F_DO_2_mod_9 : WORD ;	//error safety output 2 module 9
   error_F_DO_3_mod_9 : WORD ;	//error safety output 3 module 9
   error_F_DO_4_mod_9 : WORD ;	//error safety output 4 module 9
   error_F_Mod_R48_mod_9 : WORD ;	//error safety R48 module 9
   error_F_Mod_R49_mod_9 : WORD ;	//error safety R49 module 9
   error_F_Mod_R50_mod_9 : WORD ;	//error safety R50 module 9
   error_F_Mod_R51_mod_9 : WORD ;	//error safety R51 module 9
   error_F_Mod_R52_mod_9 : WORD ;	//error safety R52 module 9
   error_F_Mod_R53_mod_9 : WORD ;	//error safety R53 module 9
   error_F_Mod_R54_mod_9 : WORD ;	//error safety R54 module 9
   error_F_Mod_R55_mod_9 : WORD ;	//error safety R55 module 9
   F_Per_DB_B3_mod_9 : WORD ;	//state F-Periphery DB module 9
   spare_810 : WORD ;
   spare_812 : WORD ;
   spare_814 : WORD ;
   spare_816 : WORD ;
   spare_818 : WORD ;
   cmdCtrl_FB101_10 : WORD ;	//cmd / ctrl information FB101
   comCountStart_10 : WORD ;	//comCountStart indication
   mod_type_10 : WORD ;	//module type
   mod_version_10 : WORD ;	//module version
   spare_828 : WORD ;
   state_SFB52_10 : DWORD ;	//state SFB52 module
   spare_834 : WORD ;
   spare_836 : WORD ;
   error_date_mod_10 : DATE ;	//error date module 10
   error_time_mod_10 : TIME_OF_DAY ;	//error time module 10
   error_info_mod_10 : WORD ;	//error info read values module 10
   error_F_Module_mod_10 : WORD ;	//error safety module module 10
   error_F_DI_1_mod_10 : WORD ;	//error safety input 1 module 10
   error_F_DI_2_mod_10 : WORD ;	//error safety input 2 module 10
   error_F_DI_3_mod_10 : WORD ;	//error safety input 3 module 10
   error_F_DI_4_mod_10 : WORD ;	//error safety input 4 module 10
   error_F_DI_5_mod_10 : WORD ;	//error safety input 5 module 10
   error_F_DI_6_mod_10 : WORD ;	//error safety input 6 module 10
   error_F_DI_7_mod_10 : WORD ;	//error safety input 7 module 10
   error_F_DI_8_mod_10 : WORD ;	//error safety input 8 module 10
   error_F_DO_1_mod_10 : WORD ;	//error safety output 1 module 10
   error_F_DO_2_mod_10 : WORD ;	//error safety output 2 module 10
   error_F_DO_3_mod_10 : WORD ;	//error safety output 3 module 10
   error_F_DO_4_mod_10 : WORD ;	//error safety output 4 module 10
   error_F_Mod_R48_mod_10 : WORD ;	//error safety R48 module 10
   error_F_Mod_R49_mod_10 : WORD ;	//error safety R49 module 10
   error_F_Mod_R50_mod_10 : WORD ;	//error safety R50 module 10
   error_F_Mod_R51_mod_10 : WORD ;	//error safety R51 module 10
   error_F_Mod_R52_mod_10 : WORD ;	//error safety R52 module 10
   error_F_Mod_R53_mod_10 : WORD ;	//error safety R53 module 10
   error_F_Mod_R54_mod_10 : WORD ;	//error safety R54 module 10
   error_F_Mod_R55_mod_10 : WORD ;	//error safety R55 module 10
   F_Per_DB_B3_mod_10 : WORD ;	//state F-Periphery DB module 10
   spare_890 : WORD ;
   spare_892 : WORD ;
   spare_894 : WORD ;
   spare_896 : WORD ;
   spare_898 : WORD ;
   cmdCtrl_FB101_11 : WORD ;	//cmd / ctrl information FB101
   comCountStart_11 : WORD ;	//comCountStart indication
   mod_type_11 : WORD ;	//module type
   mod_version_11 : WORD ;	//module version
   spare_909 : WORD ;
   state_SFB52_11 : DWORD ;	//state SFB52 module
   spare_914 : WORD ;
   spare_916 : WORD ;
   error_date_mod_11 : DATE ;	//error date module 11
   error_time_mod_11 : TIME_OF_DAY ;	//error time module 11
   error_info_mod_11 : WORD ;	//error info read values module 11
   error_F_Module_mod_11 : WORD ;	//error safety module module 11
   error_F_DI_1_mod_11 : WORD ;	//error safety input 1 module 11
   error_F_DI_2_mod_11 : WORD ;	//error safety input 2 module 11
   error_F_DI_3_mod_11 : WORD ;	//error safety input 3 module 11
   error_F_DI_4_mod_11 : WORD ;	//error safety input 4 module 11
   error_F_DI_5_mod_11 : WORD ;	//error safety input 5 module 11
   error_F_DI_6_mod_11 : WORD ;	//error safety input 6 module 11
   error_F_DI_7_mod_11 : WORD ;	//error safety input 7 module 11
   error_F_DI_8_mod_11 : WORD ;	//error safety input 8 module 11
   error_F_DO_1_mod_11 : WORD ;	//error safety output 1 module 11
   error_F_DO_2_mod_11 : WORD ;	//error safety output 2 module 11
   error_F_DO_3_mod_11 : WORD ;	//error safety output 3 module 11
   error_F_DO_4_mod_11 : WORD ;	//error safety output 4 module 11
   error_F_Mod_R48_mod_11 : WORD ;	//error safety R48 module 11
   error_F_Mod_R49_mod_11 : WORD ;	//error safety R49 module 11
   error_F_Mod_R50_mod_11 : WORD ;	//error safety R50 module 11
   error_F_Mod_R51_mod_11 : WORD ;	//error safety R51 module 11
   error_F_Mod_R52_mod_11 : WORD ;	//error safety R52 module 11
   error_F_Mod_R53_mod_11 : WORD ;	//error safety R53 module 11
   error_F_Mod_R54_mod_11 : WORD ;	//error safety R54 module 11
   error_F_Mod_R55_mod_11 : WORD ;	//error safety R55 module 11
   F_Per_DB_B3_mod_11 : WORD ;	//state F-Periphery DB module 11
   spare_970 : WORD ;
   spare_972 : WORD ;
   spare_974 : WORD ;
   spare_976 : WORD ;
   spare_978 : WORD ;
   cmdCtrl_FB101_12 : WORD ;	//cmd / ctrl information FB101
   comCountStart_12 : WORD ;	//comCountStart indication
   mod_type_12 : WORD ;	//module type
   mod_version_12 : WORD ;	//module version
   spare_988 : WORD ;
   state_SFB52_12 : DWORD ;	//state SFB52 module
   spare_994 : WORD ;
   spare_996 : WORD ;
   error_date_mod_12 : DATE ;	//error date module 12
   error_time_mod_12 : TIME_OF_DAY ;	//error time module 12
   error_info_mod_12 : WORD ;	//error info read values module 12
   error_F_Module_mod_12 : WORD ;	//error safety module module 12
   error_F_DI_1_mod_12 : WORD ;	//error safety input 1 module 12
   error_F_DI_2_mod_12 : WORD ;	//error safety input 2 module 12
   error_F_DI_3_mod_12 : WORD ;	//error safety input 3 module 12
   error_F_DI_4_mod_12 : WORD ;	//error safety input 4 module 12
   error_F_DI_5_mod_12 : WORD ;	//error safety input 5 module 12
   error_F_DI_6_mod_12 : WORD ;	//error safety input 6 module 12
   error_F_DI_7_mod_12 : WORD ;	//error safety input 7 module 12
   error_F_DI_8_mod_12 : WORD ;	//error safety input 8 module 12
   error_F_DO_1_mod_12 : WORD ;	//error safety output 1 module 12
   error_F_DO_2_mod_12 : WORD ;	//error safety output 2 module 12
   error_F_DO_3_mod_12 : WORD ;	//error safety output 3 module 12
   error_F_DO_4_mod_12 : WORD ;	//error safety output 4 module 12
   error_F_Mod_R48_mod_12 : WORD ;	//error safety R48 module 12
   error_F_Mod_R49_mod_12 : WORD ;	//error safety R49 module 12
   error_F_Mod_R50_mod_12 : WORD ;	//error safety R50 module 12
   error_F_Mod_R51_mod_12 : WORD ;	//error safety R51 module 12
   error_F_Mod_R52_mod_12 : WORD ;	//error safety R52 module 12
   error_F_Mod_R53_mod_12 : WORD ;	//error safety R53 module 12
   error_F_Mod_R54_mod_12 : WORD ;	//error safety R54 module 12
   error_F_Mod_R55_mod_12 : WORD ;	//error safety R55 module 12
   F_Per_DB_B3_mod_12 : WORD ;	//state F-Periphery DB module 12
   spare_1050 : WORD ;
   spare_1052 : WORD ;
   spare_1054 : WORD ;
   spare_1056 : WORD ;
   spare_1058 : WORD ;
   actValuesStorage : INT ;	//info actual values storage
   spare_1062 : WORD ;
   spare_1064 : WORD ;
   spare_1066 : WORD ;
   spare_1068 : WORD ;
   I_Inf_module_Nb_1 : INT ;
   I_Error_date_mod_1 : DATE ;
   I_Error_time_mod_1 : TIME_OF_DAY ;
   I_Error_info_mod_1 : WORD ;
   I_Error_F_Module_mod_1 : WORD ;
   I_Error_F_DI_1_mod_1 : WORD ;
   I_Error_F_DI_2_mod_1 : WORD ;
   I_Error_F_DI_3_mod_1 : WORD ;
   I_Error_F_DI_4_mod_1 : WORD ;
   I_Error_F_DI_5_mod_1 : WORD ;
   I_Error_F_DI_6_mod_1 : WORD ;
   I_Error_F_DI_7_mod_1 : WORD ;
   I_Error_F_DI_8_mod_1 : WORD ;
   I_Error_F_DO_1_mod_1 : WORD ;
   I_Error_F_DO_2_mod_1 : WORD ;
   I_Error_F_DO_3_mod_1 : WORD ;
   I_Error_F_DO_4_mod_1 : WORD ;
   I_Error_F_Mod_R48_mod_1 : WORD ;
   I_Error_F_Mod_R49_mod_1 : WORD ;
   I_Error_F_Mod_R50_mod_1 : WORD ;
   I_Error_F_Mod_R51_mod_1 : WORD ;
   I_Error_F_Mod_R52_mod_1 : WORD ;
   I_Error_F_Mod_R53_mod_1 : WORD ;
   I_Error_F_Mod_R54_mod_1 : WORD ;
   I_Error_F_Mod_R55_mod_1 : WORD ;
   I_F_Per_DB_B3_mod_1 : WORD ;
   I_ModuleType_mod_1 : INT ;
   spare_1126 : WORD ;
   spare_1128 : WORD ;
   I_Inf_module_Nb_2 : INT ;
   I_Error_date_mod_2 : DATE ;
   I_Error_time_mod_2 : TIME_OF_DAY ;
   I_Error_info_mod_2 : WORD ;
   I_Error_F_Module_mod_2 : WORD ;
   I_Error_F_DI_1_mod_2 : WORD ;
   I_Error_F_DI_2_mod_2 : WORD ;
   I_Error_F_DI_3_mod_2 : WORD ;
   I_Error_F_DI_4_mod_2 : WORD ;
   I_Error_F_DI_5_mod_2 : WORD ;
   I_Error_F_DI_6_mod_2 : WORD ;
   I_Error_F_DI_7_mod_2 : WORD ;
   I_Error_F_DI_8_mod_2 : WORD ;
   I_Error_F_DO_1_mod_2 : WORD ;
   I_Error_F_DO_2_mod_2 : WORD ;
   I_Error_F_DO_3_mod_2 : WORD ;
   I_Error_F_DO_4_mod_2 : WORD ;
   I_Error_F_Mod_R48_mod_2 : WORD ;
   I_Error_F_Mod_R49_mod_2 : WORD ;
   I_Error_F_Mod_R50_mod_2 : WORD ;
   I_Error_F_Mod_R51_mod_2 : WORD ;
   I_Error_F_Mod_R52_mod_2 : WORD ;
   I_Error_F_Mod_R53_mod_2 : WORD ;
   I_Error_F_Mod_R54_mod_2 : WORD ;
   I_Error_F_Mod_R55_mod_2 : WORD ;
   I_F_Per_DB_B3_mod_2 : WORD ;
   I_ModuleType_mod_2 : INT ;
   spare_1186 : WORD ;
   spare_1188 : WORD ;
   I_Inf_module_Nb_3 : INT ;
   I_Error_date_mod_3 : DATE ;
   I_Error_time_mod_3 : TIME_OF_DAY ;
   I_Error_info_mod_3 : WORD ;
   I_Error_F_Module_mod_3 : WORD ;
   I_Error_F_DI_1_mod_3 : WORD ;
   I_Error_F_DI_2_mod_3 : WORD ;
   I_Error_F_DI_3_mod_3 : WORD ;
   I_Error_F_DI_4_mod_3 : WORD ;
   I_Error_F_DI_5_mod_3 : WORD ;
   I_Error_F_DI_6_mod_3 : WORD ;
   I_Error_F_DI_7_mod_3 : WORD ;
   I_Error_F_DI_8_mod_3 : WORD ;
   I_Error_F_DO_1_mod_3 : WORD ;
   I_Error_F_DO_2_mod_3 : WORD ;
   I_Error_F_DO_3_mod_3 : WORD ;
   I_Error_F_DO_4_mod_3 : WORD ;
   I_Error_F_Mod_R48_mod_3 : WORD ;
   I_Error_F_Mod_R49_mod_3 : WORD ;
   I_Error_F_Mod_R50_mod_3 : WORD ;
   I_Error_F_Mod_R51_mod_3 : WORD ;
   I_Error_F_Mod_R52_mod_3 : WORD ;
   I_Error_F_Mod_R53_mod_3 : WORD ;
   I_Error_F_Mod_R54_mod_3 : WORD ;
   I_Error_F_Mod_R55_mod_3 : WORD ;
   I_F_Per_DB_B3_mod_3 : WORD ;
   I_ModuleType_mod_3 : INT ;
   spare_1246 : WORD ;
   spare_1248 : WORD ;
   I_Inf_module_Nb_4 : INT ;
   I_Error_date_mod_4 : DATE ;
   I_Error_time_mod_4 : TIME_OF_DAY ;
   I_Error_info_mod_4 : WORD ;
   I_Error_F_Module_mod_4 : WORD ;
   I_Error_F_DI_1_mod_4 : WORD ;
   I_Error_F_DI_2_mod_4 : WORD ;
   I_Error_F_DI_3_mod_4 : WORD ;
   I_Error_F_DI_4_mod_4 : WORD ;
   I_Error_F_DI_5_mod_4 : WORD ;
   I_Error_F_DI_6_mod_4 : WORD ;
   I_Error_F_DI_7_mod_4 : WORD ;
   I_Error_F_DI_8_mod_4 : WORD ;
   I_Error_F_DO_1_mod_4 : WORD ;
   I_Error_F_DO_2_mod_4 : WORD ;
   I_Error_F_DO_3_mod_4 : WORD ;
   I_Error_F_DO_4_mod_4 : WORD ;
   I_Error_F_Mod_R48_mod_4 : WORD ;
   I_Error_F_Mod_R49_mod_4 : WORD ;
   I_Error_F_Mod_R50_mod_4 : WORD ;
   I_Error_F_Mod_R51_mod_4 : WORD ;
   I_Error_F_Mod_R52_mod_4 : WORD ;
   I_Error_F_Mod_R53_mod_4 : WORD ;
   I_Error_F_Mod_R54_mod_4 : WORD ;
   I_Error_F_Mod_R55_mod_4 : WORD ;
   I_F_Per_DB_B3_mod_4 : WORD ;
   I_ModuleType_mod_4 : INT ;
   spare_1306 : WORD ;
   spare_1308 : WORD ;
   I_Inf_module_Nb_5 : INT ;
   I_Error_date_mod_5 : DATE ;
   I_Error_time_mod_5 : TIME_OF_DAY ;
   I_Error_info_mod_5 : WORD ;
   I_Error_F_Module_mod_5 : WORD ;
   I_Error_F_DI_1_mod_5 : WORD ;
   I_Error_F_DI_2_mod_5 : WORD ;
   I_Error_F_DI_3_mod_5 : WORD ;
   I_Error_F_DI_4_mod_5 : WORD ;
   I_Error_F_DI_5_mod_5 : WORD ;
   I_Error_F_DI_6_mod_5 : WORD ;
   I_Error_F_DI_7_mod_5 : WORD ;
   I_Error_F_DI_8_mod_5 : WORD ;
   I_Error_F_DO_1_mod_5 : WORD ;
   I_Error_F_DO_2_mod_5 : WORD ;
   I_Error_F_DO_3_mod_5 : WORD ;
   I_Error_F_DO_4_mod_5 : WORD ;
   I_Error_F_Mod_R48_mod_5 : WORD ;
   I_Error_F_Mod_R49_mod_5 : WORD ;
   I_Error_F_Mod_R50_mod_5 : WORD ;
   I_Error_F_Mod_R51_mod_5 : WORD ;
   I_Error_F_Mod_R52_mod_5 : WORD ;
   I_Error_F_Mod_R53_mod_5 : WORD ;
   I_Error_F_Mod_R54_mod_5 : WORD ;
   I_Error_F_Mod_R55_mod_5 : WORD ;
   I_F_Per_DB_B3_mod_5 : WORD ;
   I_ModuleType_mod_5 : INT ;
   spare_1366 : WORD ;
   spare_1368 : WORD ;
   I_Inf_module_Nb_6 : INT ;
   I_Error_date_mod_6 : DATE ;
   I_Error_time_mod_6 : TIME_OF_DAY ;
   I_Error_info_mod_6 : WORD ;
   I_Error_F_Module_mod_6 : WORD ;
   I_Error_F_DI_1_mod_6 : WORD ;
   I_Error_F_DI_2_mod_6 : WORD ;
   I_Error_F_DI_3_mod_6 : WORD ;
   I_Error_F_DI_4_mod_6 : WORD ;
   I_Error_F_DI_5_mod_6 : WORD ;
   I_Error_F_DI_6_mod_6 : WORD ;
   I_Error_F_DI_7_mod_6 : WORD ;
   I_Error_F_DI_8_mod_6 : WORD ;
   I_Error_F_DO_1_mod_6 : WORD ;
   I_Error_F_DO_2_mod_6 : WORD ;
   I_Error_F_DO_3_mod_6 : WORD ;
   I_Error_F_DO_4_mod_6 : WORD ;
   I_Error_F_Mod_R48_mod_6 : WORD ;
   I_Error_F_Mod_R49_mod_6 : WORD ;
   I_Error_F_Mod_R50_mod_6 : WORD ;
   I_Error_F_Mod_R51_mod_6 : WORD ;
   I_Error_F_Mod_R52_mod_6 : WORD ;
   I_Error_F_Mod_R53_mod_6 : WORD ;
   I_Error_F_Mod_R54_mod_6 : WORD ;
   I_Error_F_Mod_R55_mod_6 : WORD ;
   I_F_Per_DB_B3_mod_6 : WORD ;
   I_ModuleType_mod_6 : INT ;
   spare_1426 : WORD ;
   spare_1428 : WORD ;
   I_Inf_module_Nb_7 : INT ;
   I_Error_date_mod_7 : DATE ;
   I_Error_time_mod_7 : TIME_OF_DAY ;
   I_Error_info_mod_7 : WORD ;
   I_Error_F_Module_mod_7 : WORD ;
   I_Error_F_DI_1_mod_7 : WORD ;
   I_Error_F_DI_2_mod_7 : WORD ;
   I_Error_F_DI_3_mod_7 : WORD ;
   I_Error_F_DI_4_mod_7 : WORD ;
   I_Error_F_DI_5_mod_7 : WORD ;
   I_Error_F_DI_6_mod_7 : WORD ;
   I_Error_F_DI_7_mod_7 : WORD ;
   I_Error_F_DI_8_mod_7 : WORD ;
   I_Error_F_DO_1_mod_7 : WORD ;
   I_Error_F_DO_2_mod_7 : WORD ;
   I_Error_F_DO_3_mod_7 : WORD ;
   I_Error_F_DO_4_mod_7 : WORD ;
   I_Error_F_Mod_R48_mod_7 : WORD ;
   I_Error_F_Mod_R49_mod_7 : WORD ;
   I_Error_F_Mod_R50_mod_7 : WORD ;
   I_Error_F_Mod_R51_mod_7 : WORD ;
   I_Error_F_Mod_R52_mod_7 : WORD ;
   I_Error_F_Mod_R53_mod_7 : WORD ;
   I_Error_F_Mod_R54_mod_7 : WORD ;
   I_Error_F_Mod_R55_mod_7 : WORD ;
   I_F_Per_DB_B3_mod_7 : WORD ;
   I_ModuleType_mod_7 : INT ;
   spare_1486 : WORD ;
   spare_1488 : WORD ;
   I_Inf_module_Nb_8 : INT ;
   I_Error_date_mod_8 : DATE ;
   I_Error_time_mod_8 : TIME_OF_DAY ;
   I_Error_info_mod_8 : WORD ;
   I_Error_F_Module_mod_8 : WORD ;
   I_Error_F_DI_1_mod_8 : WORD ;
   I_Error_F_DI_2_mod_8 : WORD ;
   I_Error_F_DI_3_mod_8 : WORD ;
   I_Error_F_DI_4_mod_8 : WORD ;
   I_Error_F_DI_5_mod_8 : WORD ;
   I_Error_F_DI_6_mod_8 : WORD ;
   I_Error_F_DI_7_mod_8 : WORD ;
   I_Error_F_DI_8_mod_8 : WORD ;
   I_Error_F_DO_1_mod_8 : WORD ;
   I_Error_F_DO_2_mod_8 : WORD ;
   I_Error_F_DO_3_mod_8 : WORD ;
   I_Error_F_DO_4_mod_8 : WORD ;
   I_Error_F_Mod_R48_mod_8 : WORD ;
   I_Error_F_Mod_R49_mod_8 : WORD ;
   I_Error_F_Mod_R50_mod_8 : WORD ;
   I_Error_F_Mod_R51_mod_8 : WORD ;
   I_Error_F_Mod_R52_mod_8 : WORD ;
   I_Error_F_Mod_R53_mod_8 : WORD ;
   I_Error_F_Mod_R54_mod_8 : WORD ;
   I_Error_F_Mod_R55_mod_8 : WORD ;
   I_F_Per_DB_B3_mod_8 : WORD ;
   I_ModuleType_mod_8 : INT ;
   spare_1546 : WORD ;
   spare_1548 : WORD ;
   I_Inf_module_Nb_9 : INT ;
   I_Error_date_mod_9 : DATE ;
   I_Error_time_mod_9 : TIME_OF_DAY ;
   I_Error_info_mod_9 : WORD ;
   I_Error_F_Module_mod_9 : WORD ;
   I_Error_F_DI_1_mod_9 : WORD ;
   I_Error_F_DI_2_mod_9 : WORD ;
   I_Error_F_DI_3_mod_9 : WORD ;
   I_Error_F_DI_4_mod_9 : WORD ;
   I_Error_F_DI_5_mod_9 : WORD ;
   I_Error_F_DI_6_mod_9 : WORD ;
   I_Error_F_DI_7_mod_9 : WORD ;
   I_Error_F_DI_8_mod_9 : WORD ;
   I_Error_F_DO_1_mod_9 : WORD ;
   I_Error_F_DO_2_mod_9 : WORD ;
   I_Error_F_DO_3_mod_9 : WORD ;
   I_Error_F_DO_4_mod_9 : WORD ;
   I_Error_F_Mod_R48_mod_9 : WORD ;
   I_Error_F_Mod_R49_mod_9 : WORD ;
   I_Error_F_Mod_R50_mod_9 : WORD ;
   I_Error_F_Mod_R51_mod_9 : WORD ;
   I_Error_F_Mod_R52_mod_9 : WORD ;
   I_Error_F_Mod_R53_mod_9 : WORD ;
   I_Error_F_Mod_R54_mod_9 : WORD ;
   I_Error_F_Mod_R55_mod_9 : WORD ;
   I_F_Per_DB_B3_mod_9 : WORD ;
   I_ModuleType_mod_9 : INT ;
   spare_1606 : WORD ;
   spare_1608 : WORD ;
   I_Inf_module_Nb_10 : INT ;
   I_Error_date_mod_10 : DATE ;
   I_Error_time_mod_10 : TIME_OF_DAY ;
   I_Error_info_mod_10 : WORD ;
   I_Error_F_Module_mod_10 : WORD ;
   I_Error_F_DI_1_mod_10 : WORD ;
   I_Error_F_DI_2_mod_10 : WORD ;
   I_Error_F_DI_3_mod_10 : WORD ;
   I_Error_F_DI_4_mod_10 : WORD ;
   I_Error_F_DI_5_mod_10 : WORD ;
   I_Error_F_DI_6_mod_10 : WORD ;
   I_Error_F_DI_7_mod_10 : WORD ;
   I_Error_F_DI_8_mod_10 : WORD ;
   I_Error_F_DO_1_mod_10 : WORD ;
   I_Error_F_DO_2_mod_10 : WORD ;
   I_Error_F_DO_3_mod_10 : WORD ;
   I_Error_F_DO_4_mod_10 : WORD ;
   I_Error_F_Mod_R48_mod_10 : WORD ;
   I_Error_F_Mod_R49_mod_10 : WORD ;
   I_Error_F_Mod_R50_mod_10 : WORD ;
   I_Error_F_Mod_R51_mod_10 : WORD ;
   I_Error_F_Mod_R52_mod_10 : WORD ;
   I_Error_F_Mod_R53_mod_10 : WORD ;
   I_Error_F_Mod_R54_mod_10 : WORD ;
   I_Error_F_Mod_R55_mod_10 : WORD ;
   I_F_Per_DB_B3_mod_10 : WORD ;
   I_ModuleType_mod_10 : INT ;
   spare_1666 : WORD ;
   spare_1668 : WORD ;
   I_Inf_module_Nb_11 : INT ;
   I_Error_date_mod_11 : DATE ;
   I_Error_time_mod_11 : TIME_OF_DAY ;
   I_Error_info_mod_11 : WORD ;
   I_Error_F_Module_mod_11 : WORD ;
   I_Error_F_DI_1_mod_11 : WORD ;
   I_Error_F_DI_2_mod_11 : WORD ;
   I_Error_F_DI_3_mod_11 : WORD ;
   I_Error_F_DI_4_mod_11 : WORD ;
   I_Error_F_DI_5_mod_11 : WORD ;
   I_Error_F_DI_6_mod_11 : WORD ;
   I_Error_F_DI_7_mod_11 : WORD ;
   I_Error_F_DI_8_mod_11 : WORD ;
   I_Error_F_DO_1_mod_11 : WORD ;
   I_Error_F_DO_2_mod_11 : WORD ;
   I_Error_F_DO_3_mod_11 : WORD ;
   I_Error_F_DO_4_mod_11 : WORD ;
   I_Error_F_Mod_R48_mod_11 : WORD ;
   I_Error_F_Mod_R49_mod_11 : WORD ;
   I_Error_F_Mod_R50_mod_11 : WORD ;
   I_Error_F_Mod_R51_mod_11 : WORD ;
   I_Error_F_Mod_R52_mod_11 : WORD ;
   I_Error_F_Mod_R53_mod_11 : WORD ;
   I_Error_F_Mod_R54_mod_11 : WORD ;
   I_Error_F_Mod_R55_mod_11 : WORD ;
   I_F_Per_DB_B3_mod_11 : WORD ;
   I_ModuleType_mod_11 : INT ;
   spare_1726 : WORD ;
   spare_1728 : WORD ;
   I_Inf_module_Nb_12 : INT ;
   I_Error_date_mod_12 : DATE ;
   I_Error_time_mod_12 : TIME_OF_DAY ;
   I_Error_info_mod_12 : WORD ;
   I_Error_F_Module_mod_12 : WORD ;
   I_Error_F_DI_1_mod_12 : WORD ;
   I_Error_F_DI_2_mod_12 : WORD ;
   I_Error_F_DI_3_mod_12 : WORD ;
   I_Error_F_DI_4_mod_12 : WORD ;
   I_Error_F_DI_5_mod_12 : WORD ;
   I_Error_F_DI_6_mod_12 : WORD ;
   I_Error_F_DI_7_mod_12 : WORD ;
   I_Error_F_DI_8_mod_12 : WORD ;
   I_Error_F_DO_1_mod_12 : WORD ;
   I_Error_F_DO_2_mod_12 : WORD ;
   I_Error_F_DO_3_mod_12 : WORD ;
   I_Error_F_DO_4_mod_12 : WORD ;
   I_Error_F_Mod_R48_mod_12 : WORD ;
   I_Error_F_Mod_R49_mod_12 : WORD ;
   I_Error_F_Mod_R50_mod_12 : WORD ;
   I_Error_F_Mod_R51_mod_12 : WORD ;
   I_Error_F_Mod_R52_mod_12 : WORD ;
   I_Error_F_Mod_R53_mod_12 : WORD ;
   I_Error_F_Mod_R54_mod_12 : WORD ;
   I_Error_F_Mod_R55_mod_12 : WORD ;
   I_F_Per_DB_B3_mod_12 : WORD ;
   I_ModuleType_mod_12 : INT ;
   spare_1782 : WORD ;
   spare_1788 : WORD ;
   I_Inf_module_Nb_13 : INT ;
   I_Error_date_mod_13 : DATE ;
   I_Error_time_mod_13 : TIME_OF_DAY ;
   I_Error_info_mod_13 : WORD ;
   I_Error_F_Module_mod_13 : WORD ;
   I_Error_F_DI_1_mod_13 : WORD ;
   I_Error_F_DI_2_mod_13 : WORD ;
   I_Error_F_DI_3_mod_13 : WORD ;
   I_Error_F_DI_4_mod_13 : WORD ;
   I_Error_F_DI_5_mod_13 : WORD ;
   I_Error_F_DI_6_mod_13 : WORD ;
   I_Error_F_DI_7_mod_13 : WORD ;
   I_Error_F_DI_8_mod_13 : WORD ;
   I_Error_F_DO_1_mod_13 : WORD ;
   I_Error_F_DO_2_mod_13 : WORD ;
   I_Error_F_DO_3_mod_13 : WORD ;
   I_Error_F_DO_4_mod_13 : WORD ;
   I_Error_F_Mod_R48_mod_13 : WORD ;
   I_Error_F_Mod_R49_mod_13 : WORD ;
   I_Error_F_Mod_R50_mod_13 : WORD ;
   I_Error_F_Mod_R51_mod_13 : WORD ;
   I_Error_F_Mod_R52_mod_13 : WORD ;
   I_Error_F_Mod_R53_mod_13 : WORD ;
   I_Error_F_Mod_R54_mod_13 : WORD ;
   I_Error_F_Mod_R55_mod_13 : WORD ;
   I_F_Per_DB_B3_mod_13 : WORD ;
   I_ModuleType_mod_13 : INT ;
   spare_1846 : WORD ;
   spare_1848 : WORD ;
   I_Inf_module_Nb_14 : INT ;
   I_Error_date_mod_14 : DATE ;
   I_Error_time_mod_14 : TIME_OF_DAY ;
   I_Error_info_mod_14 : WORD ;
   I_Error_F_Module_mod_14 : WORD ;
   I_Error_F_DI_1_mod_14 : WORD ;
   I_Error_F_DI_2_mod_14 : WORD ;
   I_Error_F_DI_3_mod_14 : WORD ;
   I_Error_F_DI_4_mod_14 : WORD ;
   I_Error_F_DI_5_mod_14 : WORD ;
   I_Error_F_DI_6_mod_14 : WORD ;
   I_Error_F_DI_7_mod_14 : WORD ;
   I_Error_F_DI_8_mod_14 : WORD ;
   I_Error_F_DO_1_mod_14 : WORD ;
   I_Error_F_DO_2_mod_14 : WORD ;
   I_Error_F_DO_3_mod_14 : WORD ;
   I_Error_F_DO_4_mod_14 : WORD ;
   I_Error_F_Mod_R48_mod_14 : WORD ;
   I_Error_F_Mod_R49_mod_14 : WORD ;
   I_Error_F_Mod_R50_mod_14 : WORD ;
   I_Error_F_Mod_R51_mod_14 : WORD ;
   I_Error_F_Mod_R52_mod_14 : WORD ;
   I_Error_F_Mod_R53_mod_14 : WORD ;
   I_Error_F_Mod_R54_mod_14 : WORD ;
   I_Error_F_Mod_R55_mod_14 : WORD ;
   I_F_Per_DB_B3_mod_14 : WORD ;
   I_ModuleType_mod_14 : INT ;
   spare_1906 : WORD ;
   spare_1908 : WORD ;
   I_Inf_module_Nb_15 : INT ;
   I_Error_date_mod_15 : DATE ;
   I_Error_time_mod_15 : TIME_OF_DAY ;
   I_Error_info_mod_15 : WORD ;
   I_Error_F_Module_mod_15 : WORD ;
   I_Error_F_DI_1_mod_15 : WORD ;
   I_Error_F_DI_2_mod_15 : WORD ;
   I_Error_F_DI_3_mod_15 : WORD ;
   I_Error_F_DI_4_mod_15 : WORD ;
   I_Error_F_DI_5_mod_15 : WORD ;
   I_Error_F_DI_6_mod_15 : WORD ;
   I_Error_F_DI_7_mod_15 : WORD ;
   I_Error_F_DI_8_mod_15 : WORD ;
   I_Error_F_DO_1_mod_15 : WORD ;
   I_Error_F_DO_2_mod_15 : WORD ;
   I_Error_F_DO_3_mod_15 : WORD ;
   I_Error_F_DO_4_mod_15 : WORD ;
   I_Error_F_Mod_R48_mod_15 : WORD ;
   I_Error_F_Mod_R49_mod_15 : WORD ;
   I_Error_F_Mod_R50_mod_15 : WORD ;
   I_Error_F_Mod_R51_mod_15 : WORD ;
   I_Error_F_Mod_R52_mod_15 : WORD ;
   I_Error_F_Mod_R53_mod_15 : WORD ;
   I_Error_F_Mod_R54_mod_15 : WORD ;
   I_Error_F_Mod_R55_mod_15 : WORD ;
   I_F_Per_DB_B3_mod_15 : WORD ;
   I_ModuleType_mod_15 : INT ;
   spare_1966 : WORD ;
   spare_1968 : WORD ;
   I_Inf_module_Nb_16 : INT ;
   I_Error_date_mod_16 : DATE ;
   I_Error_time_mod_16 : TIME_OF_DAY ;
   I_Error_info_mod_16 : WORD ;
   I_Error_F_Module_mod_16 : WORD ;
   I_Error_F_DI_1_mod_16 : WORD ;
   I_Error_F_DI_2_mod_16 : WORD ;
   I_Error_F_DI_3_mod_16 : WORD ;
   I_Error_F_DI_4_mod_16 : WORD ;
   I_Error_F_DI_5_mod_16 : WORD ;
   I_Error_F_DI_6_mod_16 : WORD ;
   I_Error_F_DI_7_mod_16 : WORD ;
   I_Error_F_DI_8_mod_16 : WORD ;
   I_Error_F_DO_1_mod_16 : WORD ;
   I_Error_F_DO_2_mod_16 : WORD ;
   I_Error_F_DO_3_mod_16 : WORD ;
   I_Error_F_DO_4_mod_16 : WORD ;
   I_Error_F_Mod_R48_mod_16 : WORD ;
   I_Error_F_Mod_R49_mod_16 : WORD ;
   I_Error_F_Mod_R50_mod_16 : WORD ;
   I_Error_F_Mod_R51_mod_16 : WORD ;
   I_Error_F_Mod_R52_mod_16 : WORD ;
   I_Error_F_Mod_R53_mod_16 : WORD ;
   I_Error_F_Mod_R54_mod_16 : WORD ;
   I_Error_F_Mod_R55_mod_16 : WORD ;
   I_F_Per_DB_B3_mod_16 : WORD ;
   I_ModuleType_mod_16 : INT ;
   spare_2026 : WORD ;
   spare_2028 : WORD ;
   I_Inf_module_Nb_17 : INT ;
   I_Error_date_mod_17 : DATE ;
   I_Error_time_mod_17 : TIME_OF_DAY ;
   I_Error_info_mod_17 : WORD ;
   I_Error_F_Module_mod_17 : WORD ;
   I_Error_F_DI_1_mod_17 : WORD ;
   I_Error_F_DI_2_mod_17 : WORD ;
   I_Error_F_DI_3_mod_17 : WORD ;
   I_Error_F_DI_4_mod_17 : WORD ;
   I_Error_F_DI_5_mod_17 : WORD ;
   I_Error_F_DI_6_mod_17 : WORD ;
   I_Error_F_DI_7_mod_17 : WORD ;
   I_Error_F_DI_8_mod_17 : WORD ;
   I_Error_F_DO_1_mod_17 : WORD ;
   I_Error_F_DO_2_mod_17 : WORD ;
   I_Error_F_DO_3_mod_17 : WORD ;
   I_Error_F_DO_4_mod_17 : WORD ;
   I_Error_F_Mod_R48_mod_17 : WORD ;
   I_Error_F_Mod_R49_mod_17 : WORD ;
   I_Error_F_Mod_R50_mod_17 : WORD ;
   I_Error_F_Mod_R51_mod_17 : WORD ;
   I_Error_F_Mod_R52_mod_17 : WORD ;
   I_Error_F_Mod_R53_mod_17 : WORD ;
   I_Error_F_Mod_R54_mod_17 : WORD ;
   I_Error_F_Mod_R55_mod_17 : WORD ;
   I_F_Per_DB_B3_mod_17 : WORD ;
   I_ModuleType_mod_17 : INT ;
   spare_2086 : WORD ;
   spare_2088 : WORD ;
   I_Inf_module_Nb_18 : INT ;
   I_Error_date_mod_18 : DATE ;
   I_Error_time_mod_18 : TIME_OF_DAY ;
   I_Error_info_mod_18 : WORD ;
   I_Error_F_Module_mod_18 : WORD ;
   I_Error_F_DI_1_mod_18 : WORD ;
   I_Error_F_DI_2_mod_18 : WORD ;
   I_Error_F_DI_3_mod_18 : WORD ;
   I_Error_F_DI_4_mod_18 : WORD ;
   I_Error_F_DI_5_mod_18 : WORD ;
   I_Error_F_DI_6_mod_18 : WORD ;
   I_Error_F_DI_7_mod_18 : WORD ;
   I_Error_F_DI_8_mod_18 : WORD ;
   I_Error_F_DO_1_mod_18 : WORD ;
   I_Error_F_DO_2_mod_18 : WORD ;
   I_Error_F_DO_3_mod_18 : WORD ;
   I_Error_F_DO_4_mod_18 : WORD ;
   I_Error_F_Mod_R48_mod_18 : WORD ;
   I_Error_F_Mod_R49_mod_18 : WORD ;
   I_Error_F_Mod_R50_mod_18 : WORD ;
   I_Error_F_Mod_R51_mod_18 : WORD ;
   I_Error_F_Mod_R52_mod_18 : WORD ;
   I_Error_F_Mod_R53_mod_18 : WORD ;
   I_Error_F_Mod_R54_mod_18 : WORD ;
   I_Error_F_Mod_R55_mod_18 : WORD ;
   I_F_Per_DB_B3_mod_18 : WORD ;
   I_ModuleType_mod_18 : INT ;
   spare_2146 : WORD ;
   spare_2148 : WORD ;
   I_Inf_module_Nb_19 : INT ;
   I_Error_date_mod_19 : DATE ;
   I_Error_time_mod_19 : TIME_OF_DAY ;
   I_Error_info_mod_19 : WORD ;
   I_Error_F_Module_mod_19 : WORD ;
   I_Error_F_DI_1_mod_19 : WORD ;
   I_Error_F_DI_2_mod_19 : WORD ;
   I_Error_F_DI_3_mod_19 : WORD ;
   I_Error_F_DI_4_mod_19 : WORD ;
   I_Error_F_DI_5_mod_19 : WORD ;
   I_Error_F_DI_6_mod_19 : WORD ;
   I_Error_F_DI_7_mod_19 : WORD ;
   I_Error_F_DI_8_mod_19 : WORD ;
   I_Error_F_DO_1_mod_19 : WORD ;
   I_Error_F_DO_2_mod_19 : WORD ;
   I_Error_F_DO_3_mod_19 : WORD ;
   I_Error_F_DO_4_mod_19 : WORD ;
   I_Error_F_Mod_R48_mod_19 : WORD ;
   I_Error_F_Mod_R49_mod_19 : WORD ;
   I_Error_F_Mod_R50_mod_19 : WORD ;
   I_Error_F_Mod_R51_mod_19 : WORD ;
   I_Error_F_Mod_R52_mod_19 : WORD ;
   I_Error_F_Mod_R53_mod_19 : WORD ;
   I_Error_F_Mod_R54_mod_19 : WORD ;
   I_Error_F_Mod_R55_mod_19 : WORD ;
   I_F_Per_DB_B3_mod_19 : WORD ;
   I_ModuleType_mod_19 : INT ;
   spare_2206 : WORD ;
   spare_2208 : WORD ;
   I_Inf_module_Nb_20 : INT ;
   I_Error_date_mod_20 : DATE ;
   I_Error_time_mod_20 : TIME_OF_DAY ;
   I_Error_info_mod_20 : WORD ;
   I_Error_F_Module_mod_20 : WORD ;
   I_Error_F_DI_1_mod_20 : WORD ;
   I_Error_F_DI_2_mod_20 : WORD ;
   I_Error_F_DI_3_mod_20 : WORD ;
   I_Error_F_DI_4_mod_20 : WORD ;
   I_Error_F_DI_5_mod_20 : WORD ;
   I_Error_F_DI_6_mod_20 : WORD ;
   I_Error_F_DI_7_mod_20 : WORD ;
   I_Error_F_DI_8_mod_20 : WORD ;
   I_Error_F_DO_1_mod_20 : WORD ;
   I_Error_F_DO_2_mod_20 : WORD ;
   I_Error_F_DO_3_mod_20 : WORD ;
   I_Error_F_DO_4_mod_20 : WORD ;
   I_Error_F_Mod_R48_mod_20 : WORD ;
   I_Error_F_Mod_R49_mod_20 : WORD ;
   I_Error_F_Mod_R50_mod_20 : WORD ;
   I_Error_F_Mod_R51_mod_20 : WORD ;
   I_Error_F_Mod_R52_mod_20 : WORD ;
   I_Error_F_Mod_R53_mod_20 : WORD ;
   I_Error_F_Mod_R54_mod_20 : WORD ;
   I_Error_F_Mod_R55_mod_20 : WORD ;
   I_F_Per_DB_B3_mod_20 : WORD ;
   I_ModuleType_mod_20 : INT ;
   spare_2266 : WORD ;
   spare_2268 : WORD ;
  END_STRUCT ;	
BEGIN
   versionInfo_1 := 101;
   versionInfo_2 := W#16#100;
   fctReqTimeout := 6000;
   dsvLength := 20;
   maxModules := 1;
END_DATA_BLOCK

DATA_BLOCK "DB_Vorlage"	// DB 999
VERSION : 0.1
  STRUCT
   _DINT : STRUCT
    _000 : DINT ;
    _001 : DINT ;
    _002 : DINT ;
    _003 : DINT ;
    _004 : DINT ;
    _005 : DINT ;
    _006 : DINT ;
    _007 : DINT ;
    _008 : DINT ;
    _009 : DINT ;
    _010 : DINT ;
    _011 : DINT ;
    _012 : DINT ;
    _013 : DINT ;
    _014 : DINT ;
    _015 : DINT ;
    _016 : DINT ;
    _017 : DINT ;
    _018 : DINT ;
    _019 : DINT ;
    _020 : DINT ;
    _021 : DINT ;
    _022 : DINT ;
    _023 : DINT ;
    _024 : DINT ;
    _025 : DINT ;
    _026 : DINT ;
    _027 : DINT ;
    _028 : DINT ;
    _029 : DINT ;
    _030 : DINT ;
    _031 : DINT ;
    _032 : DINT ;
    _033 : DINT ;
    _034 : DINT ;
    _035 : DINT ;
    _036 : DINT ;
    _037 : DINT ;
    _038 : DINT ;
    _039 : DINT ;
    _040 : DINT ;
    _041 : DINT ;
    _042 : DINT ;
    _043 : DINT ;
    _044 : DINT ;
    _045 : DINT ;
    _046 : DINT ;
    _047 : DINT ;
    _048 : DINT ;
    _049 : DINT ;
    _050 : DINT ;
    _051 : DINT ;
    _052 : DINT ;
    _053 : DINT ;
    _054 : DINT ;
    _055 : DINT ;
    _056 : DINT ;
    _057 : DINT ;
    _058 : DINT ;
    _059 : DINT ;
    _060 : DINT ;
    _061 : DINT ;
    _062 : DINT ;
    _063 : DINT ;
    _064 : DINT ;
    _065 : DINT ;
    _066 : DINT ;
    _067 : DINT ;
    _068 : DINT ;
    _069 : DINT ;
    _070 : DINT ;
    _071 : DINT ;
    _072 : DINT ;
    _073 : DINT ;
    _074 : DINT ;
    _075 : DINT ;
    _076 : DINT ;
    _077 : DINT ;
    _078 : DINT ;
    _079 : DINT ;
    _080 : DINT ;
    _081 : DINT ;
    _082 : DINT ;
    _083 : DINT ;
    _084 : DINT ;
    _085 : DINT ;
    _086 : DINT ;
    _087 : DINT ;
    _088 : DINT ;
    _089 : DINT ;
    _090 : DINT ;
    _091 : DINT ;
    _092 : DINT ;
    _093 : DINT ;
    _094 : DINT ;
    _095 : DINT ;
    _096 : DINT ;
    _097 : DINT ;
    _098 : DINT ;
    _099 : DINT ;
    _100 : DINT ;
    _101 : DINT ;
    _102 : DINT ;
    _103 : DINT ;
    _104 : DINT ;
    _105 : DINT ;
    _106 : DINT ;
    _107 : DINT ;
    _108 : DINT ;
    _109 : DINT ;
    _110 : DINT ;
    _111 : DINT ;
    _112 : DINT ;
    _113 : DINT ;
    _114 : DINT ;
    _115 : DINT ;
    _116 : DINT ;
    _117 : DINT ;
    _118 : DINT ;
    _119 : DINT ;
    _120 : DINT ;
    _121 : DINT ;
    _122 : DINT ;
    _123 : DINT ;
    _124 : DINT ;
    _125 : DINT ;
    _126 : DINT ;
    _127 : DINT ;
    _128 : DINT ;
    _129 : DINT ;
    _130 : DINT ;
    _131 : DINT ;
    _132 : DINT ;
    _133 : DINT ;
    _134 : DINT ;
    _135 : DINT ;
    _136 : DINT ;
    _137 : DINT ;
    _138 : DINT ;
    _139 : DINT ;
    _140 : DINT ;
    _141 : DINT ;
    _142 : DINT ;
    _143 : DINT ;
    _144 : DINT ;
    _145 : DINT ;
    _146 : DINT ;
    _147 : DINT ;
    _148 : DINT ;
    _149 : DINT ;
    _150 : DINT ;
    _151 : DINT ;
    _152 : DINT ;
    _153 : DINT ;
    _154 : DINT ;
    _155 : DINT ;
    _156 : DINT ;
    _157 : DINT ;
    _158 : DINT ;
    _159 : DINT ;
   END_STRUCT ;
   _INT : STRUCT
    _000 : INT ;
    _001 : INT ;
    _002 : INT ;
    _003 : INT ;
    _004 : INT ;
    _005 : INT ;
    _006 : INT ;
    _007 : INT ;
    _008 : INT ;
    _009 : INT ;
    _010 : INT ;
    _011 : INT ;
    _012 : INT ;
    _013 : INT ;
    _014 : INT ;
    _015 : INT ;
    _016 : INT ;
    _017 : INT ;
    _018 : INT ;
    _019 : INT ;
    _020 : INT ;
    _021 : INT ;
    _022 : INT ;
    _023 : INT ;
    _024 : INT ;
    _025 : INT ;
    _026 : INT ;
    _027 : INT ;
    _028 : INT ;
    _029 : INT ;
    _030 : INT ;
    _031 : INT ;
    _032 : INT ;
    _033 : INT ;
    _034 : INT ;
    _035 : INT ;
    _036 : INT ;
    _037 : INT ;
    _038 : INT ;
    _039 : INT ;
    _040 : INT ;
    _041 : INT ;
    _042 : INT ;
    _043 : INT ;
    _044 : INT ;
    _045 : INT ;
    _046 : INT ;
    _047 : INT ;
    _048 : INT ;
    _049 : INT ;
    _050 : INT ;
    _051 : INT ;
    _052 : INT ;
    _053 : INT ;
    _054 : INT ;
    _055 : INT ;
    _056 : INT ;
    _057 : INT ;
    _058 : INT ;
    _059 : INT ;
    _060 : INT ;
    _061 : INT ;
    _062 : INT ;
    _063 : INT ;
    _064 : INT ;
    _065 : INT ;
    _066 : INT ;
    _067 : INT ;
    _068 : INT ;
    _069 : INT ;
    _070 : INT ;
    _071 : INT ;
    _072 : INT ;
    _073 : INT ;
    _074 : INT ;
    _075 : INT ;
    _076 : INT ;
    _077 : INT ;
    _078 : INT ;
    _079 : INT ;
    _080 : INT ;
    _081 : INT ;
    _082 : INT ;
    _083 : INT ;
    _084 : INT ;
    _085 : INT ;
    _086 : INT ;
    _087 : INT ;
    _088 : INT ;
    _089 : INT ;
    _090 : INT ;
    _091 : INT ;
    _092 : INT ;
    _093 : INT ;
    _094 : INT ;
    _095 : INT ;
    _096 : INT ;
    _097 : INT ;
    _098 : INT ;
    _099 : INT ;
    _100 : INT ;
    _101 : INT ;
    _102 : INT ;
    _103 : INT ;
    _104 : INT ;
    _105 : INT ;
    _106 : INT ;
    _107 : INT ;
    _108 : INT ;
    _109 : INT ;
    _110 : INT ;
    _111 : INT ;
    _112 : INT ;
    _113 : INT ;
    _114 : INT ;
    _115 : INT ;
    _116 : INT ;
    _117 : INT ;
    _118 : INT ;
    _119 : INT ;
    _120 : INT ;
    _121 : INT ;
    _122 : INT ;
    _123 : INT ;
    _124 : INT ;
    _125 : INT ;
    _126 : INT ;
    _127 : INT ;
    _128 : INT ;
    _129 : INT ;
    _130 : INT ;
    _131 : INT ;
    _132 : INT ;
    _133 : INT ;
    _134 : INT ;
    _135 : INT ;
    _136 : INT ;
    _137 : INT ;
    _138 : INT ;
    _139 : INT ;
    _140 : INT ;
    _141 : INT ;
    _142 : INT ;
    _143 : INT ;
    _144 : INT ;
    _145 : INT ;
    _146 : INT ;
    _147 : INT ;
    _148 : INT ;
    _149 : INT ;
    _150 : INT ;
    _151 : INT ;
    _152 : INT ;
    _153 : INT ;
    _154 : INT ;
    _155 : INT ;
    _156 : INT ;
    _157 : INT ;
    _158 : INT ;
    _159 : INT ;
   END_STRUCT ;
   _BOOL : STRUCT
    _000 : BOOL ;
    _001 : BOOL ;
    _002 : BOOL ;
    _003 : BOOL ;
    _004 : BOOL ;
    _005 : BOOL ;
    _006 : BOOL ;
    _007 : BOOL ;
    _008 : BOOL ;
    _009 : BOOL ;
    _010 : BOOL ;
    _011 : BOOL ;
    _012 : BOOL ;
    _013 : BOOL ;
    _014 : BOOL ;
    _015 : BOOL ;
    _016 : BOOL ;
    _017 : BOOL ;
    _018 : BOOL ;
    _019 : BOOL ;
    _020 : BOOL ;
    _021 : BOOL ;
    _022 : BOOL ;
    _023 : BOOL ;
    _024 : BOOL ;
    _025 : BOOL ;
    _026 : BOOL ;
    _027 : BOOL ;
    _028 : BOOL ;
    _029 : BOOL ;
    _030 : BOOL ;
    _031 : BOOL ;
    _032 : BOOL ;
    _033 : BOOL ;
    _034 : BOOL ;
    _035 : BOOL ;
    _036 : BOOL ;
    _037 : BOOL ;
    _038 : BOOL ;
    _039 : BOOL ;
    _040 : BOOL ;
    _041 : BOOL ;
    _042 : BOOL ;
    _043 : BOOL ;
    _044 : BOOL ;
    _045 : BOOL ;
    _046 : BOOL ;
    _047 : BOOL ;
    _048 : BOOL ;
    _049 : BOOL ;
    _050 : BOOL ;
    _051 : BOOL ;
    _052 : BOOL ;
    _053 : BOOL ;
    _054 : BOOL ;
    _055 : BOOL ;
    _056 : BOOL ;
    _057 : BOOL ;
    _058 : BOOL ;
    _059 : BOOL ;
    _060 : BOOL ;
    _061 : BOOL ;
    _062 : BOOL ;
    _063 : BOOL ;
    _064 : BOOL ;
    _065 : BOOL ;
    _066 : BOOL ;
    _067 : BOOL ;
    _068 : BOOL ;
    _069 : BOOL ;
    _070 : BOOL ;
    _071 : BOOL ;
    _072 : BOOL ;
    _073 : BOOL ;
    _074 : BOOL ;
    _075 : BOOL ;
    _076 : BOOL ;
    _077 : BOOL ;
    _078 : BOOL ;
    _079 : BOOL ;
    _080 : BOOL ;
    _081 : BOOL ;
    _082 : BOOL ;
    _083 : BOOL ;
    _084 : BOOL ;
    _085 : BOOL ;
    _086 : BOOL ;
    _087 : BOOL ;
    _088 : BOOL ;
    _089 : BOOL ;
    _090 : BOOL ;
    _091 : BOOL ;
    _092 : BOOL ;
    _093 : BOOL ;
    _094 : BOOL ;
    _095 : BOOL ;
    _096 : BOOL ;
    _097 : BOOL ;
    _098 : BOOL ;
    _099 : BOOL ;
    _100 : BOOL ;
    _101 : BOOL ;
    _102 : BOOL ;
    _103 : BOOL ;
    _104 : BOOL ;
    _105 : BOOL ;
    _106 : BOOL ;
    _107 : BOOL ;
    _108 : BOOL ;
    _109 : BOOL ;
    _110 : BOOL ;
    _111 : BOOL ;
    _112 : BOOL ;
    _113 : BOOL ;
    _114 : BOOL ;
    _115 : BOOL ;
    _116 : BOOL ;
    _117 : BOOL ;
    _118 : BOOL ;
    _119 : BOOL ;
    _120 : BOOL ;
    _121 : BOOL ;
    _122 : BOOL ;
    _123 : BOOL ;
    _124 : BOOL ;
    _125 : BOOL ;
    _126 : BOOL ;
    _127 : BOOL ;
    _128 : BOOL ;
    _129 : BOOL ;
    _130 : BOOL ;
    _131 : BOOL ;
    _132 : BOOL ;
    _133 : BOOL ;
    _134 : BOOL ;
    _135 : BOOL ;
    _136 : BOOL ;
    _137 : BOOL ;
    _138 : BOOL ;
    _139 : BOOL ;
    _140 : BOOL ;
    _141 : BOOL ;
    _142 : BOOL ;
    _143 : BOOL ;
    _144 : BOOL ;
    _145 : BOOL ;
    _146 : BOOL ;
    _147 : BOOL ;
    _148 : BOOL ;
    _149 : BOOL ;
    _150 : BOOL ;
    _151 : BOOL ;
    _152 : BOOL ;
    _153 : BOOL ;
    _154 : BOOL ;
    _155 : BOOL ;
    _156 : BOOL ;
    _157 : BOOL ;
    _158 : BOOL ;
    _159 : BOOL ;
   END_STRUCT ;
  END_STRUCT ;	
BEGIN
END_DATA_BLOCK

DATA_BLOCK "DB_LS1"	// DB 1300
VERSION : 0.1
  STRUCT
   Release : STRUCT
    x_Release_From_RBG : BOOL ;
    x_Release_To_RBG : BOOL ;
    x_Chain_forward : BOOL ;
    x_Chain_backward : BOOL ;
    x_Center_Open : BOOL ;
    x_Center_Close : BOOL ;
    SPARE : ARRAY  [0 .. 9 ] OF BYTE ;
   END_STRUCT ;
   Cyl_IN : STRUCT
    x_Next : BOOL ;
    x_ToEnd : BOOL ;
    x_NextStep : BOOL ;
    x_Active : BOOL ;
    x_Finished : BOOL ;
    x_Ready : BOOL ;
    x_Start : BOOL ;
    x_Cyl_PUT : BOOL ;	//Cylinder is loaded from operator
    x_Cyl_GET : BOOL ;	//Cylinder is picked up from RBG
    x_New_Data : BOOL ;	//New cylinder data from master
    x_SPARE2 : BOOL ;
    x_SPARE3 : BOOL ;
    x_SPARE4 : BOOL ;
    x_SPARE5 : BOOL ;
    x_SPARE6 : BOOL ;
    x_SPARE7 : BOOL ;
    i_Step : INT ;
   END_STRUCT ;
   Cyl_OUT : STRUCT
    x_Next : BOOL ;
    x_ToEnd : BOOL ;
    x_NextStep : BOOL ;
    x_Active : BOOL ;
    x_Finished : BOOL ;
    x_Ready : BOOL ;
    x_Start : BOOL ;
    x_Cyl_PUT : BOOL ;	//Cylinder is loaded from RBG
    x_Cyl_GET : BOOL ;	//Cylinder is picked up from operator
    x_New_Data : BOOL ;	//New cylinder data from master
    x_SPARE2 : BOOL ;
    x_SPARE3 : BOOL ;
    x_SPARE4 : BOOL ;
    x_SPARE5 : BOOL ;
    x_SPARE6 : BOOL ;
    x_SPARE7 : BOOL ;
    i_Step : INT ;
   END_STRUCT ;
   Control : STRUCT
    x_P_Edge_FrontPos : BOOL ;
    x_P_Edge_BackPos : BOOL ;
    x_P_Edge_FNextPos : BOOL ;
    x_P_Edge_BNextPos : BOOL ;
    x_P_Edge_SPARE4 : BOOL ;
    x_P_Edge_SPARE5 : BOOL ;
    x_P_Edge_SPARE6 : BOOL ;
    x_P_Edge_SPARE7 : BOOL ;
    x_FrontPos : BOOL ;
    x_BackPos : BOOL ;
    x_Next_BackPos : BOOL ;
    x_Next_FrontPos : BOOL ;
    SPARE : ARRAY  [0 .. 99 ] OF BYTE ;
   END_STRUCT ;
   Error : STRUCT
    x_Cyl_Lentgh : BOOL ;
    x_Cyl_Circum : BOOL ;
    x_Cyl_Type : BOOL ;
    SPARE : ARRAY  [0 .. 9 ] OF BYTE ;
   END_STRUCT ;
   Order : STRUCT
    SourceBri : INT ;
    SourceTro : INT ;
    SourceLif : INT ;
    SourceTel : INT ;
    TargetBri : INT ;
    TargetTro : INT ;
    TargetLif : INT ;
    TargetTel : INT ;
    OrderTotalLength : INT ;
    OrderFaceLength : INT ;
    OrderCircum : INT ;
    ReleaseManual : BOOL ;
    spare01 : BOOL ;
    StartOrder : BOOL ;
    CleareOrder : BOOL ;
    StopOrder : BOOL ;
    spare05 : BOOL ;
    spare06 : BOOL ;
    ReleaseOnline : BOOL ;
    Lifebit : BOOL ;
    spare11 : BOOL ;
    StartBasePos : BOOL ;
    ChangeOrder : BOOL ;
    QuitOrderFinished : BOOL ;
    ResetErrors : BOOL ;
    ServiceOn : BOOL ;
    BypassLimmitsOn : BOOL ;
    SPARE : ARRAY  [0 .. 11 ] OF BYTE ;
   END_STRUCT ;
   Centering : STRUCT
    x_BtnPlus_Rais : BOOL ;
    x_BtnMinus_Rais : BOOL ;
    x_BtnPlus_RaisB : BOOL ;
    x_BtnMinus_RaisB : BOOL ;
    x_SPARE_4 : BOOL ;
    x_SPARE_5 : BOOL ;
    x_SPARE_6 : BOOL ;
    x_SPARE_7 : BOOL ;
    x_SPARE_8 : BOOL ;
    x_SPARE_9 : BOOL ;
    x_SPARE_10 : BOOL ;
    x_SPARE_11 : BOOL ;
    x_SPARE_12 : BOOL ;
    x_SPARE_13 : BOOL ;
    x_SPARE_14 : BOOL ;
    x_SPARE_15 : BOOL ;
    di_ActPos : DINT ;
    i_ActPos : INT ;
    i_ActPosNo : INT ;
    i_TargetPos : INT ;
    Positions : ARRAY  [0 .. 9 ] OF INT ;
    SPARE : ARRAY  [0 .. 11 ] OF BYTE ;
   END_STRUCT ;
   Measuring : STRUCT
    ActTotalLength : INT ;
    ActDiamterCyl : INT ;
    ActCircumCyl : INT ;
    ActValueMeasureDiameter : INT ;
    SPARE : ARRAY  [0 .. 11 ] OF BYTE ;
   END_STRUCT ;
   _di : STRUCT
    SWS_Min : DINT ;
    SWS_Max : DINT ;
    SPARE : ARRAY  [0 .. 20 ] OF DINT ;
   END_STRUCT ;
  END_STRUCT ;	
BEGIN
   Release.x_Release_From_RBG := TRUE;
   Release.x_Release_To_RBG := TRUE;
   Release.x_Chain_forward := TRUE;
   Release.x_Chain_backward := TRUE;
   Release.x_Center_Open := TRUE;
   Release.x_Center_Close := TRUE;
   Cyl_IN.x_Start := TRUE;
   Cyl_IN.x_New_Data := TRUE;
   Cyl_OUT.x_ToEnd := TRUE;
   Cyl_OUT.x_NextStep := TRUE;
   Cyl_OUT.x_Ready := TRUE;
   Cyl_OUT.x_Cyl_GET := TRUE;
   Order.OrderTotalLength := 2285;
   Order.OrderCircum := 467;
   Order.SPARE[0] := B#16#24;
   Order.SPARE[1] := B#16#40;
   Centering.di_ActPos := L#1686;
   Centering.i_ActPos := 1686;
   Centering.i_ActPosNo := 3;
   Centering.i_TargetPos := 1684;
   Centering.Positions[1] := 1579;
   Centering.Positions[2] := 1634;
   Centering.Positions[3] := 1684;
   Centering.Positions[4] := 1704;
   Centering.Positions[5] := 1804;
   Measuring.ActValueMeasureDiameter := 289;
   _di.SWS_Min := L#1625;
   _di.SWS_Max := L#1810;
END_DATA_BLOCK

DATA_BLOCK "IDB_LS1_Circum"	// DB 1329
VERSION : 0.0
"WAGO_Analog_Input_4_20"
BEGIN
END_DATA_BLOCK

DATA_BLOCK "DB_LS"	// DB 1350
VERSION : 0.1
  STRUCT
   LS1 : STRUCT
    Cart_in_Station : BOOL ;
    Hooks_02_Free : BOOL ;
    Hooks_12_Free : BOOL ;
    SPARE_03 : BOOL ;
    SPARE_04 : BOOL ;
    SPARE_05 : BOOL ;
    SPARE_06 : BOOL ;
    SPARE_07 : BOOL ;
    SPARE_10 : BOOL ;
    SPARE_11 : BOOL ;
    SPARE_12 : BOOL ;
    SPARE_13 : BOOL ;
    SPARE_14 : BOOL ;
    SPARE_15 : BOOL ;
    SPARE_16 : BOOL ;
    SPARE_17 : BOOL ;
    SPARE : ARRAY  [0 .. 12 ] OF WORD ;
   END_STRUCT ;
   LS2 : STRUCT
    Cart_in_Station : BOOL ;
    Hooks_02_Free : BOOL ;
    Hooks_12_Free : BOOL ;
    SPARE_03 : BOOL ;
    SPARE_04 : BOOL ;
    SPARE_05 : BOOL ;
    SPARE_06 : BOOL ;
    SPARE_07 : BOOL ;
    SPARE_10 : BOOL ;
    SPARE_11 : BOOL ;
    SPARE_12 : BOOL ;
    SPARE_13 : BOOL ;
    SPARE_14 : BOOL ;
    SPARE_15 : BOOL ;
    SPARE_16 : BOOL ;
    SPARE_17 : BOOL ;
    SPARE : ARRAY  [0 .. 12 ] OF WORD ;
   END_STRUCT ;
   LS3 : STRUCT
    Cart_in_Station : BOOL ;
    Hooks_02_Free : BOOL ;
    Hooks_12_Free : BOOL ;
    SPARE_03 : BOOL ;
    SPARE_04 : BOOL ;
    SPARE_05 : BOOL ;
    SPARE_06 : BOOL ;
    SPARE_07 : BOOL ;
    SPARE_10 : BOOL ;
    SPARE_11 : BOOL ;
    SPARE_12 : BOOL ;
    SPARE_13 : BOOL ;
    SPARE_14 : BOOL ;
    SPARE_15 : BOOL ;
    SPARE_16 : BOOL ;
    SPARE_17 : BOOL ;
    SPARE : ARRAY  [0 .. 12 ] OF WORD ;
   END_STRUCT ;
  END_STRUCT ;	
BEGIN
END_DATA_BLOCK

DATA_BLOCK "iPar_Data_Rack"	// DB 1901
TITLE = Vorlage Datenbaustein zur Ablage der iParameter für FB37
//Template data block used in combination with FB37
//
AUTHOR : JPR
FAMILY : WAGOiPar
NAME : iParUDL4
VERSION : 5.1
  STRUCT
   versionInfo_1 : INT  := 37;	//version info main
   versionInfo_2 : WORD  := W#16#501;	//version info release
   chkInfoData : WORD ;	//check info data
   fctReqTimeout : INT  := 6000;	//function request timeout (default 6000; av.cycle plc 5 ms - timeout 30 s)
   maxModules : INT  := 1;	//amount PROFIsafe modules FB41
   type_module_1 : INT ;	//type module 1 (661/662/663/666/667/669)
   adr_module_1 : INT ;	//I/O address module 1
   bussystem_mod_1 : INT ;	//used bussystem module 1 (0 = DP / 1 = PN)
   type_module_2 : INT ;	//type module 2 (661/662/663/666/667/669)
   adr_module_2 : INT ;	//I/O address module 2
   bussystem_mod_2 : INT ;	//used bussystem module 2 (0 = DP / 1 = PN)
   type_module_3 : INT ;	//type module 3 (661/662/663/666/667/669)
   adr_module_3 : INT ;	//I/O address module 3
   bussystem_mod_3 : INT ;	//used bussystem module 3 (0 = DP / 1 = PN)
   type_module_4 : INT ;	//type module 4 (661/662/663/666/667/669)
   adr_module_4 : INT ;	//I/O address module 4
   bussystem_mod_4 : INT ;	//used bussystem module 4 (0 = DP / 1 = PN)
   spare_34 : WORD ;
   spare_36 : WORD ;
   spare_38 : WORD ;
   spare_40 : WORD ;
   spare_42 : WORD ;
   spare_44 : WORD ;
   spare_46 : WORD ;
   spare_48 : WORD ;
   spare_50 : WORD ;
   spare_52 : WORD ;
   spare_54 : WORD ;
   spare_56 : WORD ;
   spare_58 : WORD ;
   spare_60 : WORD ;
   spare_62 : WORD ;
   spare_64 : WORD ;
   spare_66 : WORD ;
   spare_68 : WORD ;
   spare_70 : WORD ;
   spare_72 : WORD ;
   spare_74 : WORD ;
   spare_76 : WORD ;
   spare_78 : WORD ;
   spare_80 : WORD ;
   resFctReq_ok : DWORD ;	//response function request ok - "bit per module"
   resFctReq_error : DWORD ;	//response function request error - "bit per module"
   startupDate : DATE ;	//startup date application slave
   startupTime : TIME_OF_DAY ;	//startup time application slave
   slaveConfigInfo : DWORD ;	//info available PROFIsafe modules at slave
   QBAD_moduleActive : DWORD ;	//info QBAD at PROFIsafe module active
   ACK_REQ_moduleActive : DWORD ;	//info ACK_REQ at PROFIsafe module active
   READ_DIAG_REQ_module : DWORD ;	//info READ_DIAG_REQ at PROFIsafe module active
   init_fb_done : DWORD ;	//info init FB done
   check_cfg_done : DWORD ;	//info check cfg done
   upload_done : DWORD ;	//info upload slave done
   download_done : DWORD ;	//info download slave done
   compare_done : DWORD ;	//info compare slave done
   actDateCyle : DATE ;	//actual system date of cycle
   actTimeCyle : TIME_OF_DAY ;	//actual system time of cycle
   cmdCtrl_FB37 : WORD ;	//cmd / ctrl information FB37
   comCountStart_1 : WORD ;	//comCountStart indication 1
   mod_type_1 : WORD ;	//module type 1
   mod_version_1 : WORD ;	//module version 1
   spare_146 : WORD ;
   spare_148 : WORD ;
   upl_date_mod_1 : DATE ;	//upload date module 1
   upl_time_mod_1 : TIME_OF_DAY ;	//upload time module 1
   dnl_date_mod_1 : DATE ;	//download date module 1
   dnl_time_mod_1 : TIME_OF_DAY ;	//download time module 1
   cmp_date_mod_1 : DATE ;	//compare date module 1
   cmp_time_mod_1 : TIME_OF_DAY ;	//compare time module 1
   dsv_info_mod_1 : WORD ;	//dataset info module 1
   data_0_mod_1 : WORD ;	//data 0 - 1 module 1
   data_2_mod_1 : WORD ;	//data 2 - 3 module 1
   data_4_mod_1 : WORD ;	//data 4 - 5 module 1
   data_6_mod_1 : WORD ;	//data 6 - 7 module 1
   data_8_mod_1 : WORD ;	//data 8 - 9 module 1
   data_10_mod_1 : WORD ;	//data 10 - 11 module 1
   data_12_mod_1 : WORD ;	//data 12 - 13 module 1
   data_14_mod_1 : WORD ;	//data 14 - 15 module 1
   data_16_mod_1 : WORD ;	//data 16 - 17 module 1
   data_18_mod_1 : WORD ;	//data 18 - 19 module 1
   data_20_mod_1 : WORD ;	//data 20 - 21 module 1
   data_22_mod_1 : WORD ;	//data 22 - 23 module 1
   data_24_mod_1 : WORD ;	//data 24 - 25 module 1
   data_26_mod_1 : WORD ;	//data 26 - 27 module 1
   data_28_mod_1 : WORD ;	//data 28 - 29 module 1
   data_30_mod_1 : WORD ;	//data 30 - 31 module 1
   data_32_mod_1 : WORD ;	//data 32 - 33 module 1
   data_34_mod_1 : WORD ;	//data 34 - 35 module 1
   data_36_mod_1 : WORD ;	//data 36 - 37 module 1
   data_38_mod_1 : WORD ;	//data 38 - 39 module 1
   spare_210 : WORD ;
   spare_212 : WORD ;
   spare_214 : WORD ;
   spare_216 : WORD ;
   spare_218 : WORD ;
   error_Com_1 : WORD ;	//error indication  Com  module 1
   error_nb_Com_1 : WORD ;	//error number indication  Com  module 1
   state_SFB52a_1 : WORD ;	//state SFB52 part 1 module 1
   state_SFB52b_1 : WORD ;	//state SFB52 part 2 module 1
   state_SFB53a_1 : WORD ;	//state SFB53 part 1 module 1
   state_SFB53b_1 : WORD ;	//state SFB53 part 2 module 1
   spare_232 : WORD ;
   error_date_mod_1 : DATE ;	//error date module 1
   error_time_mod_1 : TIME_OF_DAY ;	//error time module 1
   error_info_mod_1 : WORD ;	//error info read values module 1
   error_F_Module_mod_1 : WORD ;	//error safety module module 1
   error_F_DI_1_mod_1 : WORD ;	//error safety input 1 module 1
   error_F_DI_2_mod_1 : WORD ;	//error safety input 2 module 1
   error_F_DI_3_mod_1 : WORD ;	//error safety input 3 module 1
   error_F_DI_4_mod_1 : WORD ;	//error safety input 4 module 1
   error_F_DI_5_mod_1 : WORD ;	//error safety input 5 module 1
   error_F_DI_6_mod_1 : WORD ;	//error safety input 6 module 1
   error_F_DI_7_mod_1 : WORD ;	//error safety input 7 module 1
   error_F_DI_8_mod_1 : WORD ;	//error safety input 8 module 1
   error_F_DO_1_mod_1 : WORD ;	//error safety output 1 module 1
   error_F_DO_2_mod_1 : WORD ;	//error safety output 2 module 1
   error_F_DO_3_mod_1 : WORD ;	//error safety output 3 module 1
   error_F_DO_4_mod_1 : WORD ;	//error safety output 4 module 1
   error_Reg52_mod_1 : WORD ;	//error safety module register 52 module 1
   error_Reg53_mod_1 : WORD ;	//error safety module register 53 module 1
   error_Reg54_mod_1 : WORD ;	//error safety module register 54 module 1
   error_Reg55_mod_1 : WORD ;	//error safety module register 55 module 1
   spare_276 : WORD ;
   spare_278 : WORD ;
   comCountStart_2 : WORD ;	//comCountStart indication 2
   mod_type_2 : WORD ;	//module type 2
   mod_version_2 : WORD ;	//module version 2
   spare_286 : WORD ;
   spare_288 : WORD ;
   upl_date_mod_2 : DATE ;	//upload date module 2
   upl_time_mod_2 : TIME_OF_DAY ;	//upload time module 2
   dnl_date_mod_2 : DATE ;	//download date module 2
   dnl_time_mod_2 : TIME_OF_DAY ;	//download time module 2
   cmp_date_mod_2 : DATE ;	//compare date module 2
   cmp_time_mod_2 : TIME_OF_DAY ;	//compare time module 2
   dsv_info_mod_2 : WORD ;	//dataset info module 2
   data_0_mod_2 : WORD ;	//data 0 - 1 module 2
   data_2_mod_2 : WORD ;	//data 2 - 3 module 2
   data_4_mod_2 : WORD ;	//data 4 - 5 module 2
   data_6_mod_2 : WORD ;	//data 6 - 7 module 2
   data_8_mod_2 : WORD ;	//data 8 - 9 module 2
   data_10_mod_2 : WORD ;	//data 10 - 11 module 2
   data_12_mod_2 : WORD ;	//data 12 - 13 module 2
   data_14_mod_2 : WORD ;	//data 14 - 15 module 2
   data_16_mod_2 : WORD ;	//data 16 - 17 module 2
   data_18_mod_2 : WORD ;	//data 18 - 19 module 2
   data_20_mod_2 : WORD ;	//data 20 - 21 module 2
   data_22_mod_2 : WORD ;	//data 22 - 23 module 2
   data_24_mod_2 : WORD ;	//data 24 - 25 module 2
   data_26_mod_2 : WORD ;	//data 26 - 27 module 2
   data_28_mod_2 : WORD ;	//data 28 - 29 module 2
   data_30_mod_2 : WORD ;	//data 30 - 31 module 2
   data_32_mod_2 : WORD ;	//data 32 - 33 module 2
   data_34_mod_2 : WORD ;	//data 34 - 35 module 2
   data_36_mod_2 : WORD ;	//data 36 - 37 module 2
   data_38_mod_2 : WORD ;	//data 38 - 39 module 2
   spare_350 : WORD ;
   spare_352 : WORD ;
   spare_354 : WORD ;
   spare_356 : WORD ;
   spare_358 : WORD ;
   error_Com_2 : WORD ;	//error indication  Com  module 2
   error_nb_Com_2 : WORD ;	//error number indication  Com  module 2
   state_SFB52a_2 : WORD ;	//state SFB52 part 1 module 2
   state_SFB52b_2 : WORD ;	//state SFB52 part 2 module 2
   state_SFB53a_2 : WORD ;	//state SFB53 part 1 module 2
   state_SFB53b_2 : WORD ;	//state SFB53 part 2 module 2
   spare_372 : WORD ;
   error_date_mod_2 : DATE ;	//error date module 2
   error_time_mod_2 : TIME_OF_DAY ;	//error time module 2
   error_info_mod_2 : WORD ;	//error info read values module 2
   error_F_Module_mod_2 : WORD ;	//error safety module module 2
   error_F_DI_1_mod_2 : WORD ;	//error safety input 1 module 2
   error_F_DI_2_mod_2 : WORD ;	//error safety input 2 module 2
   error_F_DI_3_mod_2 : WORD ;	//error safety input 3 module 2
   error_F_DI_4_mod_2 : WORD ;	//error safety input 4 module 2
   error_F_DI_5_mod_2 : WORD ;	//error safety input 5 module 2
   error_F_DI_6_mod_2 : WORD ;	//error safety input 6 module 2
   error_F_DI_7_mod_2 : WORD ;	//error safety input 7 module 2
   error_F_DI_8_mod_2 : WORD ;	//error safety input 8 module 2
   error_F_DO_1_mod_2 : WORD ;	//error safety output 1 module 2
   error_F_DO_2_mod_2 : WORD ;	//error safety output 2 module 2
   error_F_DO_3_mod_2 : WORD ;	//error safety output 3 module 2
   error_F_DO_4_mod_2 : WORD ;	//error safety output 4 module 2
   error_Reg52_mod_2 : WORD ;	//error safety module register 52 module 2
   error_Reg53_mod_2 : WORD ;	//error safety module register 53 module 2
   error_Reg54_mod_2 : WORD ;	//error safety module register 54 module 2
   error_Reg55_mod_2 : WORD ;	//error safety module register 55 module 2
   spare_416 : WORD ;
   spare_418 : WORD ;
   comCountStart_3 : WORD ;	//comCountStart indication 3
   mod_type_3 : WORD ;	//module type 3
   mod_version_3 : WORD ;	//module version 3
   spare_426 : WORD ;
   spare_428 : WORD ;
   upl_date_mod_3 : DATE ;	//upload date module 3
   upl_time_mod_3 : TIME_OF_DAY ;	//upload time module 3
   dnl_date_mod_3 : DATE ;	//download date module 3
   dnl_time_mod_3 : TIME_OF_DAY ;	//download time module 3
   cmp_date_mod_3 : DATE ;	//compare date module  3
   cmp_time_mod_3 : TIME_OF_DAY ;	//compare time module  3
   dsv_info_mod_3 : WORD ;	//dataset info module 3
   data_0_mod_3 : WORD ;	//data 0 - 1 module 3
   data_2_mod_3 : WORD ;	//data 2 - 3 module 3
   data_4_mod_3 : WORD ;	//data 4 - 5 module 3
   data_6_mod_3 : WORD ;	//data 6 - 7 module 3
   data_8_mod_3 : WORD ;	//data 8 - 9 module 3
   data_10_mod_3 : WORD ;	//data 10 - 11 module 3
   data_12_mod_3 : WORD ;	//data 12 - 13 module 3
   data_14_mod_3 : WORD ;	//data 14 - 15 module 3
   data_16_mod_3 : WORD ;	//data 16 - 17 module 3
   data_18_mod_3 : WORD ;	//data 18 - 19 module 3
   data_20_mod_3 : WORD ;	//data 20 - 21 module 3
   data_22_mod_3 : WORD ;	//data 22 - 23 module 3
   data_24_mod_3 : WORD ;	//data 24 - 25 module 3
   data_26_mod_3 : WORD ;	//data 26 - 27 module 3
   data_28_mod_3 : WORD ;	//data 28 - 29 module 3
   data_30_mod_3 : WORD ;	//data 30 - 31 module 3
   data_32_mod_3 : WORD ;	//data 32 - 33 module 3
   data_34_mod_3 : WORD ;	//data 34 - 35 module 3
   data_36_mod_3 : WORD ;	//data 36 - 37 module 3
   data_38_mod_3 : WORD ;	//data 38 - 39 module 3
   spare_490 : WORD ;
   spare_492 : WORD ;
   spare_494 : WORD ;
   spare_496 : WORD ;
   spare_498 : WORD ;
   error_Com_3 : WORD ;	//error indication  Com  module 3
   error_nb_Com_3 : WORD ;	//error number indication  Com  module 3
   state_SFB52a_3 : WORD ;	//state SFB52 part 1 module 3
   state_SFB52b_3 : WORD ;	//state SFB52 part 2 module 3
   state_SFB53a_3 : WORD ;	//state SFB53 part 1 module 3
   state_SFB53b_3 : WORD ;	//state SFB53 part 2 module 3
   spare_512 : WORD ;
   error_date_mod_3 : DATE ;	//error date module 3
   error_time_mod_3 : TIME_OF_DAY ;	//error time module 3
   error_info_mod_3 : WORD ;	//error info read values module 3
   error_F_Module_mod_3 : WORD ;	//error safety module module 3
   error_F_DI_1_mod_3 : WORD ;	//error safety input 1 module 3
   error_F_DI_2_mod_3 : WORD ;	//error safety input 2 module 3
   error_F_DI_3_mod_3 : WORD ;	//error safety input 3 module 3
   error_F_DI_4_mod_3 : WORD ;	//error safety input 4 module 3
   error_F_DI_5_mod_3 : WORD ;	//error safety input 5 module 3
   error_F_DI_6_mod_3 : WORD ;	//error safety input 6 module 3
   error_F_DI_7_mod_3 : WORD ;	//error safety input 7 module 3
   error_F_DI_8_mod_3 : WORD ;	//error safety input 8 module 3
   error_F_DO_1_mod_3 : WORD ;	//error safety output 1 module 3
   error_F_DO_2_mod_3 : WORD ;	//error safety output 2 module 3
   error_F_DO_3_mod_3 : WORD ;	//error safety output 3 module 3
   error_F_DO_4_mod_3 : WORD ;	//error safety output 4 module 3
   error_Reg52_mod_3 : WORD ;	//error safety module register 52 module 3
   error_Reg53_mod_3 : WORD ;	//error safety module register 53 module 3
   error_Reg54_mod_3 : WORD ;	//error safety module register 54 module 3
   error_Reg55_mod_3 : WORD ;	//error safety module register 55 module 3
   spare_556 : WORD ;
   spare_558 : WORD ;
   comCountStart_4 : WORD ;	//comCountStart indication 4
   mod_type_4 : WORD ;	//module type  4
   mod_version_4 : WORD ;	//module version  4
   spare_566 : WORD ;
   spare_568 : WORD ;
   upl_date_mod_4 : DATE ;	//upload date module  4
   upl_time_mod_4 : TIME_OF_DAY ;	//upload time module  4
   dnl_date_mod_4 : DATE ;	//download date module  4
   dnl_time_mod_4 : TIME_OF_DAY ;	//download time module  4
   cmp_date_mod_4 : DATE ;	//compare date module   4
   cmp_time_mod_4 : TIME_OF_DAY ;	//compare time module   4
   dsv_info_mod_4 : WORD ;	//dataset info module 4
   data_0_mod_4 : WORD ;	//data 0 - 1 module  4
   data_2_mod_4 : WORD ;	//data 2 - 3 module  4
   data_4_mod_4 : WORD ;	//data 4 - 5 module  4
   data_6_mod_4 : WORD ;	//data 6 - 7 module  4
   data_8_mod_4 : WORD ;	//data 8 - 9 module  4
   data_10_mod_4 : WORD ;	//data 10 - 11 module  4
   data_12_mod_4 : WORD ;	//data 12 - 13 module  4
   data_14_mod_4 : WORD ;	//data 14 - 15 module  4
   data_16_mod_4 : WORD ;	//data 16 - 17 module  4
   data_18_mod_4 : WORD ;	//data 18 - 19 module  4
   data_20_mod_4 : WORD ;	//data 20 - 21 module  4
   data_22_mod_4 : WORD ;	//data 22 - 23 module  4
   data_24_mod_4 : WORD ;	//data 24 - 25 module  4
   data_26_mod_4 : WORD ;	//data 26 - 27 module  4
   data_28_mod_4 : WORD ;	//data 28 - 29 module  4
   data_30_mod_4 : WORD ;	//data 30 - 31 module  4
   data_32_mod_4 : WORD ;	//data 32 - 33 module  4
   data_34_mod_4 : WORD ;	//data 34 - 35 module  4
   data_36_mod_4 : WORD ;	//data 36 - 37 module  4
   data_38_mod_4 : WORD ;	//data 38 - 39 module  4
   spare_630 : WORD ;
   spare_632 : WORD ;
   spare_634 : WORD ;
   spare_636 : WORD ;
   spare_638 : WORD ;
   error_Com_4 : WORD ;	//error indication  Com  module 4
   error_nb_Com_4 : WORD ;	//error number indication  Com  module 4
   state_SFB52a_4 : WORD ;	//state SFB52 part 1 module 4
   state_SFB52b_4 : WORD ;	//state SFB52 part 2 module 4
   state_SFB53a_4 : WORD ;	//state SFB53 part 1 module 4
   state_SFB53b_4 : WORD ;	//state SFB53 part 2 module 4
   spare_652 : WORD ;
   error_date_mod_4 : DATE ;	//error date module 4
   error_time_mod_4 : TIME_OF_DAY ;	//error time module 4
   error_info_mod_4 : WORD ;	//error info read values module 4
   error_F_Module_mod_4 : WORD ;	//error safety module module 4
   error_F_DI_1_mod_4 : WORD ;	//error safety input 1 module 4
   error_F_DI_2_mod_4 : WORD ;	//error safety input 2 module 4
   error_F_DI_3_mod_4 : WORD ;	//error safety input 3 module 4
   error_F_DI_4_mod_4 : WORD ;	//error safety input 4 module 4
   error_F_DI_5_mod_4 : WORD ;	//error safety input 5 module 4
   error_F_DI_6_mod_4 : WORD ;	//error safety input 6 module 4
   error_F_DI_7_mod_4 : WORD ;	//error safety input 7 module 4
   error_F_DI_8_mod_4 : WORD ;	//error safety input 8 module 4
   error_F_DO_1_mod_4 : WORD ;	//error safety output 1 module 4
   error_F_DO_2_mod_4 : WORD ;	//error safety output 2 module 4
   error_F_DO_3_mod_4 : WORD ;	//error safety output 3 module 4
   error_F_DO_4_mod_4 : WORD ;	//error safety output 4 module 4
   error_Reg52_mod_4 : WORD ;	//error safety module register 52 module 4
   error_Reg53_mod_4 : WORD ;	//error safety module register 53 module 4
   error_Reg54_mod_4 : WORD ;	//error safety module register 54 module 4
   error_Reg55_mod_4 : WORD ;	//error safety module register 55 module 4
   spare_696 : WORD ;
   spare_698 : WORD ;
  END_STRUCT ;	
BEGIN
   versionInfo_1 := 37;
   versionInfo_2 := W#16#501;
   chkInfoData := W#16#3;
   fctReqTimeout := 6000;
   maxModules := 3;
   type_module_1 := 662;
   adr_module_1 := 40;
   bussystem_mod_1 := 1;
   type_module_2 := 667;
   adr_module_2 := 45;
   bussystem_mod_2 := 1;
   type_module_3 := 666;
   adr_module_3 := 50;
   bussystem_mod_3 := 1;
   bussystem_mod_4 := 1;
   slaveConfigInfo := DW#16#7;
   init_fb_done := DW#16#7;
   check_cfg_done := DW#16#7;
   upload_done := DW#16#7;
   download_done := DW#16#7;
   compare_done := DW#16#7;
   cmdCtrl_FB37 := W#16#FE00;
   comCountStart_1 := W#16#2;
   mod_type_1 := W#16#19E5;
   mod_version_1 := W#16#3;
   dsv_info_mod_1 := W#16#1FF0;
   data_0_mod_1 := W#16#4545;
   data_2_mod_1 := W#16#10CC;
   data_4_mod_1 := W#16#20CC;
   data_6_mod_1 := W#16#202;
   data_8_mod_1 := W#16#4FF;
   data_10_mod_1 := W#16#F;
   data_12_mod_1 := W#16#6400;
   data_14_mod_1 := W#16#6400;
   data_16_mod_1 := W#16#6400;
   data_18_mod_1 := W#16#6400;
   data_22_mod_1 := W#16#F01F;
   data_24_mod_1 := W#16#FEFF;
   data_26_mod_1 := W#16#1C72;
   data_28_mod_1 := W#16#5B54;
   data_32_mod_1 := W#16#3341;
   comCountStart_2 := W#16#2;
   mod_type_2 := W#16#1A17;
   mod_version_2 := W#16#3;
   dsv_info_mod_2 := W#16#7573;
   data_0_mod_2 := W#16#4545;
   data_2_mod_2 := W#16#10CC;
   data_4_mod_2 := W#16#20CC;
   data_6_mod_2 := W#16#203;
   data_8_mod_2 := W#16#F430;
   data_10_mod_2 := W#16#6400;
   data_12_mod_2 := W#16#6400;
   data_16_mod_2 := W#16#100;
   data_18_mod_2 := W#16#3733;
   data_20_mod_2 := W#16#7375;
   data_22_mod_2 := W#16#FEFF;
   data_24_mod_2 := W#16#B6E;
   data_26_mod_2 := W#16#5B54;
   data_30_mod_2 := W#16#7E16;
   comCountStart_3 := W#16#2;
   mod_type_3 := W#16#1A0D;
   mod_version_3 := W#16#3;
   dsv_info_mod_3 := W#16#B395;
   data_0_mod_3 := W#16#4545;
   data_2_mod_3 := W#16#10CC;
   data_4_mod_3 := W#16#20CC;
   data_6_mod_3 := W#16#204;
   data_8_mod_3 := W#16#F430;
   data_10_mod_3 := W#16#6400;
   data_12_mod_3 := W#16#6400;
   data_18_mod_3 := W#16#AA00;
   data_20_mod_3 := W#16#95B3;
   data_22_mod_3 := W#16#FEFF;
   data_24_mod_3 := W#16#CC3D;
   data_26_mod_3 := W#16#1256;
   data_30_mod_3 := W#16#E0D;
END_DATA_BLOCK

